(* IEC 61131-3 sources: ATCMcontrol_Engineering/src/COM/softing/fc/CL/Libs/ATCM_IEC1131_3, 277 files *)

(* ---- abs.st ---- *)
(*[[
    UserURL= "ATCMfile:ABS.htm"
]]*)

FUNCTION ABS : ANY_NUM
VAR_INPUT
    IN : ANY_NUM;
END_VAR

overload () inline{java.lang.Math.abs(%1)}

END_FUNCTION

(* ---- acos.st ---- *)
(*[[
    UserURL= "ATCMfile:ACOS.htm"
]]*)

FUNCTION ACOS : ANY_REAL
VAR_INPUT
    IN : ANY_REAL;
END_VAR

overload () inline{java.lang.Math.acos(%1)}

END_FUNCTION

(* ---- add.st ---- *)
(*[[
    UserURL= "ATCMFile:ADD.htm"
]]*)

FUNCTION ADD : ANY_MAGNITUDE
VAR_INPUT
    IN1 : ANY_MAGNITUDE;
END_VAR
VAR_IN_EXT
    IN2 : ANY_MAGNITUDE;
END_VAR

inline +

END_FUNCTION

(* ---- add_dt_time.st ---- *)
(*[[
    UserURL= "ATCMFile:ADD_DT_TIME.htm"
]]*)

FUNCTION ADD_DT_TIME : DT
VAR_INPUT
    IN1  : DT;
    IN2  : TIME;
END_VAR
inline +
END_FUNCTION

(* ---- add_time.st ---- *)
(*[[
    UserURL= "ATCMFile:ADD_TIME.htm"
]]*)

FUNCTION ADD_TIME : TIME
VAR_INPUT
    IN1 : TIME;
    IN2 : TIME;
END_VAR

inline +

END_FUNCTION

(* ---- add_tod_time.st ---- *)
(*[[
    UserURL= "ATCMFile:ADD_TOD_TIME.htm"
]]*)

FUNCTION ADD_TOD_TIME : TOD
VAR_INPUT
    IN1 : TOD;
    IN2 : TIME;
END_VAR
inline +
END_FUNCTION

(* ---- and.st ---- *)
(*[[
    UserURL= "ATCMFile:AND.htm"
]]*)

FUNCTION AND : ANY_BIT
VAR_INPUT
    IN1 : ANY_BIT;
END_VAR
VAR_IN_EXT
    IN2 : ANY_BIT;
END_VAR

inline AND

END_FUNCTION

(* ---- asin.st ---- *)
(*[[
    UserURL= "ATCMFile:ASIN.htm"
]]*)

FUNCTION ASIN : ANY_REAL
VAR_INPUT
    IN : ANY_REAL;
END_VAR

overload () inline{java.lang.Math.asin(%1)}

END_FUNCTION

(* ---- atan.st ---- *)
(*[[
    UserURL= "ATCMFile:ATAN.htm"
]]*)

FUNCTION ATAN : ANY_REAL
VAR_INPUT
    IN : ANY_REAL;
END_VAR

overload () inline{java.lang.Math.atan(%1)}

END_FUNCTION

(* ---- bool_to_byte.st ---- *)
(*[[
    UserURL= "ATCMFile:BOOL_TO_BYTE.htm"
]]*)

FUNCTION BOOL_TO_BYTE : BYTE
VAR_INPUT
    IN : BOOL;
END_VAR

inline{%1?1:0}

END_FUNCTION

(* ---- bool_to_dint.st ---- *)
(*[[
    UserURL= "ATCMFile:BOOL_TO_DINT.htm"
]]*)

FUNCTION BOOL_TO_DINT : DINT
VAR_INPUT
    IN : BOOL;
END_VAR

inline{%1?1:0}

END_FUNCTION

(* ---- bool_to_dword.st ---- *)
(*[[
    UserURL= "ATCMFile:BOOL_TO_DWORD.htm"
]]*)

FUNCTION BOOL_TO_DWORD : DWORD
VAR_INPUT
    IN : BOOL;
END_VAR

inline{%1?1:0}

END_FUNCTION

(* ---- bool_to_int.st ---- *)
(*[[
    UserURL= "ATCMFile:BOOL_TO_INT.htm"
]]*)

FUNCTION BOOL_TO_INT : INT
VAR_INPUT
    IN : BOOL;
END_VAR

inline{ VMOP(bool_to_int) }

END_FUNCTION

(* ---- bool_to_lint.st ---- *)
(*[[
    UserURL= "ATCMFile:BOOL_TO_LINT.htm"
]]*)

FUNCTION BOOL_TO_LINT : LINT
VAR_INPUT
    IN : BOOL;
END_VAR

inline{%1?1l:0l}

END_FUNCTION

(* ---- bool_to_lreal.st ---- *)
(*[[
    UserURL= "ATCMFile:BOOL_TO_LREAL.htm"
]]*)

FUNCTION BOOL_TO_LREAL : LREAL
VAR_INPUT
    IN : BOOL;
END_VAR

inline{%1?1.0:0.0}

END_FUNCTION

(* ---- bool_to_lword.st ---- *)
(*[[
    UserURL= "ATCMFile:BOOL_TO_LWORD.htm"
]]*)

FUNCTION BOOL_TO_LWORD : LWORD
VAR_INPUT
    IN : BOOL;
END_VAR

inline{%1?1l:0l}

END_FUNCTION

(* ---- bool_to_real.st ---- *)
(*[[
    UserURL= "ATCMFile:BOOL_TO_REAL.htm"
]]*)

FUNCTION BOOL_TO_REAL : REAL
VAR_INPUT
    IN : BOOL;
END_VAR

inline{ VMOP }

END_FUNCTION

(* ---- bool_to_string.st ---- *)
(*[[
    UserURL= "ATCMFile:BOOL_TO_STRING.htm"
]]*)

FUNCTION BOOL_TO_STRING : STRING
VAR_INPUT
    IN : BOOL;
END_VAR

inline{ STDLIB(bool_to_string) }

END_FUNCTION

(* ---- bool_to_udint.st ---- *)
(*[[
    UserURL= "ATCMFile:BOOL_TO_UDINT.htm"
]]*)
FUNCTION BOOL_TO_UDINT : UDINT
VAR_INPUT
    IN : BOOL;
END_VAR

inline{ VMOP }

END_FUNCTION

(* ---- bool_to_uint.st ---- *)
(*[[
    UserURL= "ATCMFile:BOOL_TO_UINT.htm"
]]*)
FUNCTION BOOL_TO_UINT : UINT
VAR_INPUT
    IN : BOOL;
END_VAR

inline{ VMOP }

END_FUNCTION

(* ---- bool_to_word.st ---- *)
(*[[
    UserURL= "ATCMFile:BOOL_TO_WORD.htm"
]]*)

FUNCTION BOOL_TO_WORD : WORD
VAR_INPUT
    IN : BOOL;
END_VAR

inline{%1?1:0}

END_FUNCTION

(* ---- bool_to_wstring.st ---- *)
(*[[
    UserURL= "ATCMFile:BOOL_TO_WSTRING.htm"
]]*)

FUNCTION BOOL_TO_WSTRING : WSTRING
VAR_INPUT
    IN : BOOL;
END_VAR

inline{%1?"TRUE":"FALSE"}

END_FUNCTION

(* ---- byte_to_bool.st ---- *)
(*[[
    UserURL= "ATCMFile:BYTE_TO_BOOL.htm"
]]*)

FUNCTION BYTE_TO_BOOL : BOOL
VAR_INPUT
    IN : BYTE;
END_VAR

inline{%1==0?false:true}

END_FUNCTION

(* ---- byte_to_dint.st ---- *)
(*[[
    UserURL= "ATCMFile:BYTE_TO_DINT.htm"
]]*)

FUNCTION BYTE_TO_DINT : DINT
VAR_INPUT
    IN : BYTE;
END_VAR

inline{%1}

END_FUNCTION

(* ---- byte_to_dword.st ---- *)
(*[[
    UserURL= "ATCMFile:BYTE_TO_DWORD.htm"
]]*)

FUNCTION BYTE_TO_DWORD : DWORD
VAR_INPUT
    IN : BYTE;
END_VAR

inline{%1}

END_FUNCTION

(* ---- byte_to_int.st ---- *)
(*[[
    UserURL= "ATCMFile:BYTE_TO_INT.htm"
]]*)

FUNCTION BYTE_TO_INT : INT
VAR_INPUT
    IN : BYTE;
END_VAR

inline{ VMOP }

END_FUNCTION

(* ---- byte_to_lint.st ---- *)
(*[[
    UserURL= "ATCMFile:BYTE_TO_LINT.htm"
]]*)

FUNCTION BYTE_TO_LINT : LINT
VAR_INPUT
    IN : BYTE;
END_VAR

inline{(long)%1}

END_FUNCTION

(* ---- byte_to_lreal.st ---- *)
(*[[
    UserURL= "ATCMFile:BYTE_TO_LREAL.htm"
]]*)

FUNCTION BYTE_TO_LREAL : LREAL
VAR_INPUT
    IN : BYTE;
END_VAR

inline{(double)%1}

END_FUNCTION

(* ---- byte_to_lword.st ---- *)
(*[[
    UserURL= "ATCMFile:BYTE_TO_LWORD.htm"
]]*)

FUNCTION BYTE_TO_LWORD : LWORD
VAR_INPUT
    IN : BYTE;
END_VAR

inline{(long)%1}

END_FUNCTION

(* ---- byte_to_real.st ---- *)
(*[[
    UserURL= "ATCMFile:BYTE_TO_REAL.htm"
]]*)

FUNCTION BYTE_TO_REAL : REAL
VAR_INPUT
    IN : BYTE;
END_VAR

inline{VMOP}

END_FUNCTION

(* ---- byte_to_string.st ---- *)
(*[[
    UserURL= "ATCMFile:BYTE_TO_STRING.htm"
]]*)

FUNCTION BYTE_TO_STRING : STRING
VAR_INPUT
    IN : BYTE;
END_VAR

inline{ STDLIB(byte_to_string) }

END_FUNCTION

(* ---- byte_to_udint.st ---- *)
(*[[
    UserURL= "ATCMFile:BYTE_TO_UDINT.htm"
]]*)
FUNCTION BYTE_TO_UDINT : UDINT
VAR_INPUT
    IN : BYTE;
END_VAR

inline{ VMOP }

END_FUNCTION

(* ---- byte_to_uint.st ---- *)
(*[[
    UserURL= "ATCMFile:BYTE_TO_UINT.htm"
]]*)
FUNCTION BYTE_TO_UINT : UINT
VAR_INPUT
    IN : BYTE;
END_VAR

inline{ VMOP }

END_FUNCTION

(* ---- byte_to_word.st ---- *)
(*[[
    UserURL= "ATCMFile:BYTE_TO_WORD.htm"
]]*)

FUNCTION BYTE_TO_WORD : WORD
VAR_INPUT
    IN : BYTE;
END_VAR

inline{%1}

END_FUNCTION

(* ---- byte_to_wstring.st ---- *)
(*[[
    UserURL= "ATCMFile:BYTE_TO_WSTRING.htm"
]]*)

FUNCTION BYTE_TO_WSTRING : WSTRING
VAR_INPUT
    IN : BYTE;
END_VAR

inline{java.lang.Integer.toString(%1)}

END_FUNCTION

(* ---- concat.st ---- *)
(*[[
    UserURL= "ATCMFile:CONCAT.htm"
]]*)

FUNCTION CONCAT : ANY_STRING
VAR_INPUT
    IN1 : ANY_STRING;
END_VAR
VAR_IN_EXT
    IN2 : ANY_STRING;
END_VAR

overload() inline {@+}

END_FUNCTION

(* ---- concat_date_tod.st ---- *)
(*[[
    UserURL= "ATCMFile:CONCAT_DATE_TOD.htm"
]]*)

FUNCTION CONCAT_DATE_TOD : DT
VAR_INPUT
    IN1 : DATE;
    IN2 : TOD;
END_VAR

inline{Utils.concat_date_tod(%1,%2)}

END_FUNCTION

(* ---- cos.st ---- *)
(*[[
    UserURL= "ATCMFile:COS.htm"
]]*)

FUNCTION COS : ANY_REAL
VAR_INPUT
    IN : ANY_REAL;
END_VAR

overload () inline{java.lang.Math.cos(%1)}

END_FUNCTION

(* ---- date_to_wstring.st ---- *)
(*[[
    UserURL= "ATCMFile:DATE_TO_WSTRING.htm"
]]*)

FUNCTION DATE_TO_WSTRING : WSTRING
VAR_INPUT
    IN : DATE;
END_VAR

inline{Utils.date_to_wstring(%1)}

END_FUNCTION

(* ---- delete.st ---- *)
(*[[
    UserURL= "ATCMFile:DELETE.htm"
]]*)

FUNCTION DELETE : ANY_STRING
VAR_INPUT
    IN : ANY_STRING;
    L : ANY_INT;
    P : ANY_INT;
END_VAR

overload STRING(STRING,INT,INT)
    inline{ STDLIB(DeleteString_int)}

overload STRING(STRING,DINT,DINT)
    inline{
        %res
        %2
        dint_to_int
        %3
        dint_to_int
        %1
        calfsys #DeleteString_int
		leave 8
        }

(*
overload STRING(STRING,LINT,LINT)
    inline{
        %res
        %2
        lint_to_int
        %3
        lint_to_int
        %1
        calfsys #DeleteString_int
	leave 12
        }

overload STRING(STRING,SINT,SINT)
    inline{
        %res
        %2
        sint_to_int
        %3
        sint_to_int
        %1
        calfsys #DeleteString_int
	leave 12
        }
*)

END_FUNCTION

(* ---- delete_dint.st ---- *)
(*[[
    UserURL= "ATCMFile:DELETE_DINT.htm"
]]*)

FUNCTION DELETE_DINT : ANY_STRING
VAR_INPUT
    IN : ANY_STRING;
    L  : DINT;
    P  : DINT;
END_VAR

overload() inline{Utils.deleteString(%1,%2,%3)}

END_FUNCTION

(* ---- dint_to_bool.st ---- *)
(*[[
    UserURL= "ATCMFile:DINT_TO_BOOL.htm"
]]*)

FUNCTION DINT_TO_BOOL : BOOL
VAR_INPUT
    IN : DINT;
END_VAR

inline{%1==0?false:true}

END_FUNCTION

(* ---- dint_to_byte.st ---- *)
(*[[
    UserURL= "ATCMFile:DINT_TO_BYTE.htm"
]]*)

FUNCTION DINT_TO_BYTE : BYTE
VAR_INPUT
    IN : DINT;
END_VAR

inline{%1&0xff}

END_FUNCTION

(* ---- dint_to_dword.st ---- *)
(*[[
    UserURL= "ATCMFile:DINT_TO_DWORD.htm"
]]*)

FUNCTION DINT_TO_DWORD : DWORD
VAR_INPUT
    IN : DINT;
END_VAR

inline{%1}

END_FUNCTION

(* ---- dint_to_int.st ---- *)
(*[[
    UserURL= "ATCMFile:DINT_TO_INT.htm"
]]*)

FUNCTION DINT_TO_INT : INT
VAR_INPUT
    IN : DINT;
END_VAR

inline{VMOP}

END_FUNCTION

(* ---- dint_to_lint.st ---- *)
(*[[
    UserURL= "ATCMFile:DINT_TO_LINT.htm"
]]*)

FUNCTION DINT_TO_LINT : LINT
VAR_INPUT
    IN : DINT;
END_VAR

inline{(long)%1}

END_FUNCTION

(* ---- dint_to_lreal.st ---- *)
(*[[
    UserURL= "ATCMFile:DINT_TO_LREAL.htm"
]]*)

FUNCTION DINT_TO_LREAL : LREAL
VAR_INPUT
    IN : DINT;
END_VAR

inline{(double)%1}

END_FUNCTION

(* ---- dint_to_lword.st ---- *)
(*[[
    UserURL= "ATCMFile:DINT_TO_LWORD.htm"
]]*)

FUNCTION DINT_TO_LWORD : LWORD
VAR_INPUT
    IN : DINT;
END_VAR

inline{(long)%1}

END_FUNCTION

(* ---- dint_to_real.st ---- *)
(*[[
    UserURL= "ATCMFile:DINT_TO_REAL.htm"
]]*)

FUNCTION DINT_TO_REAL : REAL
VAR_INPUT
    IN : DINT;
END_VAR

inline{VMOP}

END_FUNCTION

(* ---- dint_to_string.st ---- *)
(*[[
    UserURL= "ATCMFile:DINT_TO_STRING.htm"
]]*)

FUNCTION DINT_TO_STRING : STRING
VAR_INPUT
    IN : DINT;
END_VAR

inline{ STDLIB(dint_to_string) }

END_FUNCTION

(* ---- dint_to_time.st ---- *)
(*[[
    UserURL= "ATCMFile:DINT_TO_TIME.htm"
]]*)

FUNCTION DINT_TO_TIME : TIME
VAR_INPUT
    IN : DINT;
END_VAR

inline{(long)%1}

END_FUNCTION

(* ---- dint_to_udint.st ---- *)
(*[[
    UserURL= "ATCMFile:DINT_TO_UDINT.htm"
]]*)
FUNCTION DINT_TO_UDINT : UDINT
VAR_INPUT
    IN : DINT;
END_VAR

inline{NOOP}

END_FUNCTION

(* ---- dint_to_uint.st ---- *)
(*[[
    UserURL= "ATCMFile:DINT_TO_UINT.htm"
]]*)
FUNCTION DINT_TO_UINT : UINT
VAR_INPUT
    IN : DINT;
END_VAR

inline{ VMOP }

END_FUNCTION

(* ---- dint_to_word.st ---- *)
(*[[
    UserURL= "ATCMFile:DINT_TO_WORD.htm"
]]*)

FUNCTION DINT_TO_WORD : WORD
VAR_INPUT
    IN : DINT;
END_VAR

inline{%1&0xffff}

END_FUNCTION

(* ---- dint_to_wstring.st ---- *)
(*[[
    UserURL= "ATCMFile:DINT_TO_WSTRING.htm"
]]*)

FUNCTION DINT_TO_WSTRING : WSTRING
VAR_INPUT
    IN : DINT;
END_VAR

inline{java.lang.Integer.toString(%1)}

END_FUNCTION

(* ---- div.st ---- *)
(*[[
    UserURL= "ATCMFile:DIV.htm"
]]*)

FUNCTION DIV : ANY_NUM
VAR_INPUT
    IN1: ANY_NUM;
    IN2: ANY_NUM;
END_VAR

inline /

END_FUNCTION

(* ---- divtime.st ---- *)
(*[[
    UserURL= "ATCMFile:DIVTIME.htm"
]]*)

FUNCTION DIVTIME : TIME
VAR_INPUT
    IN1 : TIME;
    IN2 : ANY_NUM;
END_VAR

inline /

END_FUNCTION

(* ---- dt_to_date.st ---- *)
(*[[
    UserURL= "ATCMFile:DT_TO_DATE.htm"
]]*)

FUNCTION DT_TO_DATE : DATE
VAR_INPUT
    IN : DT;
END_VAR

inline{Utils.dt_to_date(%1)}

END_FUNCTION

(* ---- dt_to_time.st ---- *)
(*[[
    UserURL= "ATCMFile:DT_TO_TIME.htm"
]]*)

FUNCTION DT_TO_TIME : TIME
VAR_INPUT
    IN : DT;
END_VAR

inline{%1}

END_FUNCTION

(* ---- dt_to_tod.st ---- *)
(*[[
    UserURL= "ATCMFile:DT_TO_TOD.htm"
]]*)

FUNCTION DT_TO_TOD : TOD
VAR_INPUT
    IN : DT;
END_VAR

inline{Utils.dt_to_tod(%1)}

END_FUNCTION

(* ---- dt_to_wstring.st ---- *)
(*[[
    UserURL= "ATCMFile:DT_TO_WSTRING.htm"
]]*)

FUNCTION DT_TO_WSTRING : WSTRING
VAR_INPUT
    IN : DT;
END_VAR

inline{Utils.dt_to_wstring(%1)}

END_FUNCTION

(* ---- dword_to_bool.st ---- *)
(*[[
    UserURL= "ATCMFile:DWORD_TO_BOOL.htm"
]]*)

FUNCTION DWORD_TO_BOOL : BOOL
VAR_INPUT
    IN : DWORD;
END_VAR

inline{%1==0?false:true}

END_FUNCTION

(* ---- dword_to_byte.st ---- *)
(*[[
    UserURL= "ATCMFile:DWORD_TO_BYTE.htm"
]]*)

FUNCTION DWORD_TO_BYTE : BYTE
VAR_INPUT
    IN : DWORD;
END_VAR

inline{%1&0xff}

END_FUNCTION

(* ---- dword_to_dint.st ---- *)
(*[[
    UserURL= "ATCMFile:DWORD_TO_DINT.htm"
]]*)

FUNCTION DWORD_TO_DINT : DINT
VAR_INPUT
    IN : DWORD;
END_VAR

inline{%1}

END_FUNCTION

(* ---- dword_to_int.st ---- *)
(*[[
    UserURL= "ATCMFile:DWORD_TO_INT.htm"
]]*)

FUNCTION DWORD_TO_INT : INT
VAR_INPUT
    IN : DWORD;
END_VAR

inline{VMOP}

END_FUNCTION

(* ---- dword_to_lint.st ---- *)
(*[[
    UserURL= "ATCMFile:DWORD_TO_LINT.htm"
]]*)

FUNCTION DWORD_TO_LINT : LINT
VAR_INPUT
    IN : DWORD;
END_VAR

inline{((long)%1)&0xffffffffl}

END_FUNCTION

(* ---- dword_to_lreal.st ---- *)
(*[[
    UserURL= "ATCMFile:DWORD_TO_LREAL.htm"
]]*)

FUNCTION DWORD_TO_LREAL : LREAL
VAR_INPUT
    IN : DWORD;
END_VAR

inline{(double)(0x00000000ffffffffL & %1)}

END_FUNCTION

(* ---- dword_to_lword.st ---- *)
(*[[
    UserURL= "ATCMFile:DWORD_TO_LWORD.htm"
]]*)

FUNCTION DWORD_TO_LWORD : LWORD
VAR_INPUT
    IN : DWORD;
END_VAR

inline{((long)%1)&0xffffffffl}

END_FUNCTION

(* ---- dword_to_real.st ---- *)
(*[[
    UserURL= "ATCMFile:DWORD_TO_REAL.htm"
]]*)

FUNCTION DWORD_TO_REAL : REAL
VAR_INPUT
    IN : DWORD;
END_VAR

inline{VMOP}

END_FUNCTION

(* ---- dword_to_string.st ---- *)
(*[[
    UserURL= "ATCMFile:DWORD_TO_STRING.htm"
]]*)

FUNCTION DWORD_TO_STRING : STRING
VAR_INPUT
    IN : DWORD;
END_VAR

inline{ STDLIB(dword_to_string) }

END_FUNCTION

(* ---- dword_to_udint.st ---- *)
(*[[
    UserURL= "ATCMFile:DWORD_TO_UDINT.htm"
]]*)
FUNCTION DWORD_TO_UDINT : UDINT
VAR_INPUT
    IN : DWORD;
END_VAR

inline{NOOP}

END_FUNCTION

(* ---- dword_to_uint.st ---- *)
(*[[
    UserURL= "ATCMFile:DWORD_TO_UINT.htm"
]]*)
FUNCTION DWORD_TO_UINT : UINT
VAR_INPUT
    IN : DWORD;
END_VAR

inline{ VMOP }

END_FUNCTION

(* ---- dword_to_word.st ---- *)
(*[[
    UserURL= "ATCMFile:DWORD_TO_WORD.htm"
]]*)

FUNCTION DWORD_TO_WORD : WORD
VAR_INPUT
    IN : DWORD;
END_VAR

inline{%1&0xffff}

END_FUNCTION

(* ---- dword_to_wstring.st ---- *)
(*[[
    UserURL= "ATCMFile:DWORD_TO_WSTRING.htm"
]]*)

FUNCTION DWORD_TO_WSTRING : WSTRING
VAR_INPUT
    IN : DWORD;
END_VAR

inline{java.lang.Long.toString(0x00000000ffffffffL & %1)}

END_FUNCTION

(* ---- eq.st ---- *)
(*[[
    UserURL= "ATCMFile:EQ.htm"
]]*)

FUNCTION EQ : BOOL
VAR_INPUT
    IN1 : ANY_ELEMENTARY;
END_VAR
VAR_IN_EXT
    IN2 : ANY_ELEMENTARY;
END_VAR

inline =

END_FUNCTION

(* ---- exp.st ---- *)
(*[[
    UserURL= "ATCMFile:EXP.htm"
]]*)

FUNCTION EXP : ANY_REAL
VAR_INPUT
    IN : ANY_REAL;
END_VAR

overload () inline{java.lang.Math.exp(%1)}

END_FUNCTION

(* ---- expt.st ---- *)
(*[[
    UserURL= "ATCMFile:EXPT.htm"
]]*)

FUNCTION EXPT : ANY_REAL
VAR_INPUT
    IN1: ANY_REAL;
    IN2: ANY_NUM;
END_VAR

inline **

END_FUNCTION

(* ---- find.st ---- *)
(*[[
    UserURL= "ATCMFile:FIND.htm"
]]*)

FUNCTION FIND : ANY_INT
VAR_INPUT
    IN1 : ANY_STRING;
    IN2 : ANY_STRING;
END_VAR

overload INT(STRING,STRING)
    inline{ STDLIB(FindString_int) }

overload DINT(STRING,STRING)
    inline{
        %res
        dint_to_int
        %2
        %1
        calfsys #FindString_int
		leave 8
		int_to_dint
        }

(*
overload LINT(STRING,STRING)
    inline{
        %res
        lint_to_int
        %2
        %1
        calfsys #FindString_int
	leave 10
        }

overload SINT(STRING,STRING)
    inline{
        %res
        sint_to_int
        %2
        %1
        calfsys #FindString_int
	leave 10
        }
*)

END_FUNCTION

(* ---- find_dint.st ---- *)
(*[[
    UserURL= "ATCMFile:FIND_DINT.htm"
]]*)
FUNCTION FIND_DINT : DINT
VAR_INPUT
    IN1 : ANY_STRING;
    IN2 : ANY_STRING;
END_VAR

overload() inline{%1.indexOf(%2)+1}

END_FUNCTION

(* ---- ge.st ---- *)
(*[[
    UserURL= "ATCMFile:GE.htm"
]]*)

FUNCTION GE : BOOL
VAR_INPUT
    IN1 : ANY_ELEMENTARY;
END_VAR
VAR_IN_EXT
    IN2 : ANY_ELEMENTARY;
END_VAR

inline >=

END_FUNCTION

(* ---- gt.st ---- *)
(*[[
    UserURL= "ATCMFile:GT.htm"
]]*)

FUNCTION GT : BOOL
VAR_INPUT
    IN1 : ANY_ELEMENTARY;
END_VAR
VAR_IN_EXT
    IN2 : ANY_ELEMENTARY;
END_VAR

inline >

END_FUNCTION

(* ---- insert.st ---- *)
(*[[
    UserURL= "ATCMFile:INSERT.htm"
]]*)

FUNCTION INSERT : ANY_STRING
VAR_INPUT
    IN1 : ANY_STRING;
    IN2 : ANY_STRING;
    P : ANY_INT;
END_VAR

overload STRING(STRING,STRING,INT)
    inline{ STDLIB(InsertString_int)}

overload STRING(STRING,STRING,DINT)
    inline{
        %res
        %3
        dint_to_int
        %2
        %1
        calfsys #InsertString_int
		leave 10
        }

(*
overload STRING(STRING,STRING,LINT)
    inline{
        %res
        %3
        lint_to_int
        %2
        %1
        calfsys #InsertString_int
	leave 14
        }

overload STRING(STRING,STRING,SINT)
    inline{
        %res
        %3
        sint_to_int
        %2
        %1
        calfsys #InsertString_int
	leave 14
        }
*)

END_FUNCTION

(* ---- insert_dint.st ---- *)
(*[[
    UserURL= "ATCMFile:INSERT_DINT.htm"
]]*)

FUNCTION INSERT_DINT : ANY_STRING
VAR_INPUT
    IN1 : ANY_STRING;
    IN2 : ANY_STRING;
    P   : DINT;
END_VAR

overload() inline{Utils.insertString(%1,%2,%3)}

END_FUNCTION

(* ---- int_to_bool.st ---- *)
(*[[
    UserURL= "ATCMFile:INT_TO_BOOL.htm"
]]*)

FUNCTION INT_TO_BOOL : BOOL
VAR_INPUT
    IN : INT;
END_VAR

inline{VMOP(WORD_TO_BOOL)}

END_FUNCTION

(* ---- int_to_byte.st ---- *)
(*[[
    UserURL= "ATCMFile:INT_TO_BYTE.htm"
]]*)

FUNCTION INT_TO_BYTE : BYTE
VAR_INPUT
    IN : INT;
END_VAR

inline{VMOP(word_to_byte
; int_to_byte
; push word#16#ff
; and_word
)
      }

END_FUNCTION

(* ---- int_to_dint.st ---- *)
(*[[
    UserURL= "ATCMFile:INT_TO_DINT.htm"
]]*)

FUNCTION INT_TO_DINT : DINT
VAR_INPUT
    IN : INT;
END_VAR

inline{VMOP}

END_FUNCTION

(* ---- int_to_dword.st ---- *)
(*[[
    UserURL= "ATCMFile:INT_TO_DWORD.htm"
]]*)

FUNCTION INT_TO_DWORD : DWORD
VAR_INPUT
    IN : INT;
END_VAR

inline{VMOP}

END_FUNCTION

(* ---- int_to_lint.st ---- *)
(*[[
    UserURL= "ATCMFile:INT_TO_LINT.htm"
]]*)

FUNCTION INT_TO_LINT : LINT
VAR_INPUT
    IN : INT;
END_VAR

inline{VMOP}

END_FUNCTION

(* ---- int_to_lreal.st ---- *)
(*[[
    UserURL= "ATCMFile:INT_TO_LREAL.htm"
]]*)

FUNCTION INT_TO_LREAL : LREAL
VAR_INPUT
    IN : INT;
END_VAR

inline{VMOP}

END_FUNCTION

(* ---- int_to_real.st ---- *)
(*[[
    UserURL= "ATCMFile:INT_TO_REAL.htm"
]]*)

FUNCTION INT_TO_REAL : REAL
VAR_INPUT
    IN : INT;
END_VAR

inline{VMOP}

END_FUNCTION

(* ---- int_to_string.st ---- *)
(*[[
    UserURL= "ATCMFile:INT_TO_STRING.htm"
]]*)

FUNCTION INT_TO_STRING : STRING
VAR_INPUT
    IN : INT;
END_VAR

inline{ STDLIB(int_to_string) }

END_FUNCTION

(* ---- int_to_time.st ---- *)
(*[[
    UserURL= "ATCMFile:INT_TO_TIME.htm"
]]*)

FUNCTION INT_TO_TIME : TIME
VAR_INPUT
    IN : INT;
END_VAR

inline
{
	%1
	int_to_dint
}

END_FUNCTION

(* ---- int_to_udint.st ---- *)
(*[[
    UserURL= "ATCMFile:INT_TO_UDINT.htm"
]]*)
FUNCTION INT_TO_UDINT : UDINT
VAR_INPUT
    IN : INT;
END_VAR

inline{ VMOP }

END_FUNCTION

(* ---- int_to_uint.st ---- *)
(*[[
    UserURL= "ATCMFile:INT_TO_UINT.htm"
]]*)
FUNCTION INT_TO_UINT : UINT
VAR_INPUT
    IN : INT;
END_VAR

inline{NOOP}

END_FUNCTION

(* ---- int_to_word.st ---- *)
(*[[
    UserURL= "ATCMFile:INT_TO_WORD.htm"
]]*)

FUNCTION INT_TO_WORD : WORD
VAR_INPUT
    IN : INT;
END_VAR

inline{NOOP}

END_FUNCTION

(* ---- le.st ---- *)
(*[[
    UserURL= "ATCMFile:LE.htm"
]]*)

FUNCTION LE : BOOL
VAR_INPUT
    IN1 : ANY_ELEMENTARY;
END_VAR
VAR_IN_EXT
    IN2 : ANY_ELEMENTARY;
END_VAR

inline <=

END_FUNCTION

(* ---- left.st ---- *)
(*[[
    UserURL= "ATCMFile:LEFT.htm"
]]*)
FUNCTION LEFT : ANY_STRING
VAR_INPUT
    IN : ANY_STRING;
    L : ANY_INT;
END_VAR

overload STRING(STRING,INT)
    inline{ STDLIB(LeftString_int) }

overload STRING(STRING,DINT)
    inline{
        %res
        %2
        dint_to_int
        %1
        calfsys #LeftString_int
		leave 6
        }

(*
overload STRING(STRING,LINT)
    inline{
        %res
        %2
        lint_to_int
        %1
        calfsys #LeftString_int
        leave 10
        }

overload STRING(STRING,SINT)
    inline{
        %res
        %2
        sint_to_int
        %1
        calfsys #LeftString_int
        leave 10
        }
*)

END_FUNCTION

(* ---- left_dint.st ---- *)
(*[[
    UserURL= "ATCMFile:LEFT_DINT.htm"
]]*)

FUNCTION LEFT_DINT : ANY_STRING
VAR_INPUT
    IN : ANY_STRING;
    L  : DINT;
END_VAR

overload() inline{%1.substring(0,%2)}

END_FUNCTION

(* ---- len.st ---- *)
(*[[
    UserURL= "ATCMFile:LEN.htm"
]]*)
FUNCTION LEN : ANY_INT
VAR_INPUT
    IN : STRING;
END_VAR

overload INT(STRING) inline { STDLIB(strlen_int) }
overload DINT(STRING) inline
{
	%res
	%1
    calfsys #strlen_int %leave
    int_to_dint
}

END_FUNCTION

(* ---- len_dint.st ---- *)
(*[[
    UserURL= "ATCMFile:LEN_DINT.htm"
]]*)

FUNCTION LEN_DINT : DINT
VAR_INPUT
    IN : ANY_STRING;
END_VAR

overload() inline{%1.length()}

END_FUNCTION

(* ---- limit.st ---- *)
(*[[
    UserURL= "ATCMFile:LIMIT.htm"
]]*)

FUNCTION LIMIT : ANY_ELEMENTARY
VAR_INPUT
    MN : ANY_ELEMENTARY;
    IN : ANY_ELEMENTARY;
    MX : ANY_ELEMENTARY;
END_VAR

overload DINT|LINT|LREAL|TIME|ANY_DATE|BYTE|WORD(
         DINT|LINT|LREAL|TIME|ANY_DATE|BYTE|WORD,
         DINT|LINT|LREAL|TIME|ANY_DATE|BYTE|WORD,
         DINT|LINT|LREAL|TIME|ANY_DATE|BYTE|WORD)       inline{Math.min(Math.max(%2,%1),%3)}

overload DWORD(DWORD, DWORD, DWORD)                     inline{Utils.minDword(Utils.maxDword(%2,%1),%3)}
overload LWORD(LWORD, LWORD, LWORD)                     inline{Utils.minLword(Utils.maxLword(%2,%1),%3)}
overload ANY_STRING(ANY_STRING, ANY_STRING, ANY_STRING) inline{Utils.minString(Utils.maxString(%2,%1),%3)}
overload BOOL(BOOL, BOOL, BOOL)                         inline{(%2||%1) && %3}

END_FUNCTION

(* ---- lint_to_bool.st ---- *)
(*[[
    UserURL= "ATCMFile:LINT_TO_BOOL.htm"
]]*)

FUNCTION LINT_TO_BOOL : BOOL
VAR_INPUT
    IN : LINT;
END_VAR

inline{%1==0l?false:true}

END_FUNCTION

(* ---- lint_to_byte.st ---- *)
(*[[
    UserURL= "ATCMFile:LINT_TO_BYTE.htm"
]]*)

FUNCTION LINT_TO_BYTE : BYTE
VAR_INPUT
    IN : LINT;
END_VAR

inline{(int)%1&0xff}

END_FUNCTION

(* ---- lint_to_dint.st ---- *)
(*[[
    UserURL= "ATCMFile:LINT_TO_DINT.htm"
]]*)

FUNCTION LINT_TO_DINT : DINT
VAR_INPUT
    IN : LINT;
END_VAR

inline{(int)%1}

END_FUNCTION

(* ---- lint_to_dword.st ---- *)
(*[[
    UserURL= "ATCMFile:LINT_TO_DWORD.htm"
]]*)

FUNCTION LINT_TO_DWORD : DWORD
VAR_INPUT
    IN : LINT;
END_VAR

inline{(int)%1}

END_FUNCTION

(* ---- lint_to_int.st ---- *)
(*[[
    UserURL= "ATCMFile:LINT_TO_INT.htm"
]]*)

FUNCTION LINT_TO_INT : INT
VAR_INPUT
    IN : LINT;
END_VAR

inline{(int)%1}

END_FUNCTION

(* ---- lint_to_lreal.st ---- *)
(*[[
    UserURL= "ATCMFile:LINT_TO_LREAL.htm"
]]*)

FUNCTION LINT_TO_LREAL : LREAL
VAR_INPUT
    IN : LINT;
END_VAR

inline{(double)%1}

END_FUNCTION

(* ---- lint_to_lword.st ---- *)
(*[[
    UserURL= "ATCMFile:LINT_TO_LWORD.htm"
]]*)

FUNCTION LINT_TO_LWORD : LWORD
VAR_INPUT
    IN : LINT;
END_VAR

inline{%1}

END_FUNCTION

(* ---- lint_to_real.st ---- *)
(*[[
    UserURL= "ATCMFile:LINT_TO_REAL.htm"
]]*)

FUNCTION LINT_TO_REAL : REAL
VAR_INPUT
    IN : LINT;
END_VAR

inline{(double)%1}

END_FUNCTION

(* ---- lint_to_string.st ---- *)
(*[[
    UserURL= "ATCMFile:LINT_TO_STRING.htm"
]]*)

FUNCTION LINT_TO_STRING : STRING
VAR_INPUT
    IN : LINT;
END_VAR

inline{java.lang.Long.toString(%1)}

END_FUNCTION

(* ---- lint_to_time.st ---- *)
(*[[
    UserURL= "ATCMFile:LINT_TO_TIME.htm"
]]*)

FUNCTION LINT_TO_TIME : TIME
VAR_INPUT
    IN : LINT;
END_VAR

inline{%1}

END_FUNCTION

(* ---- lint_to_word.st ---- *)
(*[[
    UserURL= "ATCMFile:LINT_TO_WORD.htm"
]]*)

FUNCTION LINT_TO_WORD : WORD
VAR_INPUT
    IN : LINT;
END_VAR

inline{(int)%1&0xffff}

END_FUNCTION

(* ---- lint_to_wstring.st ---- *)
(*[[
    UserURL= "ATCMFile:LINT_TO_WSTRING.htm"
]]*)

FUNCTION LINT_TO_WSTRING : WSTRING
VAR_INPUT
    IN : LINT;
END_VAR

inline{java.lang.Long.toString(%1)}

END_FUNCTION

(* ---- ln.st ---- *)
(*[[
    UserURL= "ATCMFile:LN.htm"
]]*)

FUNCTION LN : ANY_REAL
VAR_INPUT
    IN : ANY_REAL;
END_VAR

overload () inline{java.lang.Math.log(%1)}

END_FUNCTION

(* ---- log.st ---- *)
(*[[
    UserURL= "ATCMFile:LOG.htm"
]]*)

FUNCTION LOG : ANY_REAL
VAR_INPUT
    IN : ANY_REAL;
END_VAR

overload () inline{java.lang.Math.log(%1)/java.lang.Math.log(10)}

END_FUNCTION

(* ---- lreal_to_bool.st ---- *)
(*[[
    UserURL= "ATCMFile:LREAL_TO_BOOL.htm"
]]*)

FUNCTION LREAL_TO_BOOL : BOOL
VAR_INPUT
    IN : LREAL;
END_VAR

inline{%1==0.0?false:true}

END_FUNCTION

(* ---- lreal_to_byte.st ---- *)
(*[[
    UserURL= "ATCMFile:LREAL_TO_BYTE.htm"
]]*)

FUNCTION LREAL_TO_BYTE : BYTE
VAR_INPUT
    IN : LREAL;
END_VAR

inline{((int)Math.round(%1))&0xff}

END_FUNCTION

(* ---- lreal_to_dint.st ---- *)
(*[[
    UserURL= "ATCMFile:LREAL_TO_DINT.htm"
]]*)

FUNCTION LREAL_TO_DINT : DINT
VAR_INPUT
    IN : LREAL;
END_VAR

inline{Utils.doubleToIntIEC599(%1)}

END_FUNCTION

(* ---- lreal_to_dword.st ---- *)
(*[[
    UserURL= "ATCMFile:LREAL_TO_DWORD.htm"
]]*)

FUNCTION LREAL_TO_DWORD : DWORD
VAR_INPUT
    IN : LREAL;
END_VAR

inline{(int)Math.round(%1)}

END_FUNCTION

(* ---- lreal_to_int.st ---- *)
(*[[
    UserURL= "ATCMFile:LREAL_TO_INT.htm"
]]*)

FUNCTION LREAL_TO_INT : INT
VAR_INPUT
    IN : LREAL;
END_VAR

inline{VMOP}

END_FUNCTION

(* ---- lreal_to_lint.st ---- *)
(*[[
    UserURL= "ATCMFile:LREAL_TO_LINT.htm"
]]*)

FUNCTION LREAL_TO_LINT : LINT
VAR_INPUT
    IN : LREAL;
END_VAR

inline{Utils.doubleToLongIEC599(%1)}

END_FUNCTION

(* ---- lreal_to_lword.st ---- *)
(*
 * Note:
 *  LREAL_TO_LWORD(x) is the same as
 *  LINT_TO_LWORD(LREAL_TO_LINT(x))
 *
 *  e.g.  LREAL_TO_LWORD(-1.0E0) = 16#ffffffffffffffff;
 *)

FUNCTION LREAL_TO_LWORD : LWORD
VAR_INPUT
    IN : LREAL;
END_VAR

inline{Math.round(%1)}

END_FUNCTION

(* ---- lreal_to_real.st ---- *)
(*[[
    UserURL= "ATCMFile:LREAL_TO_REAL.htm"
]]*)

FUNCTION LREAL_TO_REAL : REAL
VAR_INPUT
    IN : LREAL;
END_VAR

inline{VMOP}

END_FUNCTION

(* ---- lreal_to_string.st ---- *)
(*[[
    UserURL= "ATCMFile:LREAL_TO_STRING.htm"
]]*)

FUNCTION LREAL_TO_STRING : STRING
VAR_INPUT
    IN : LREAL;
END_VAR

inline{ STDLIB(lreal_to_string)}

END_FUNCTION

(* ---- lreal_to_time.st ---- *)
(*[[
    UserURL= "ATCMFile:LREAL_TO_TIME.htm"
]]*)

FUNCTION LREAL_TO_TIME : TIME
VAR_INPUT
    IN : LREAL;
END_VAR

inline{(long)%1}

END_FUNCTION

(* ---- lreal_to_udint.st ---- *)
(*[[
    UserURL= "ATCMFile:LREAL_TO_UDINT.htm"
]]*)
FUNCTION LREAL_TO_UDINT : UDINT
VAR_INPUT
    IN : LREAL;
END_VAR

inline{ VMOP }

END_FUNCTION

(* ---- lreal_to_uint.st ---- *)
(*[[
    UserURL= "ATCMFile:LREAL_TO_UINT.htm"
]]*)
FUNCTION LREAL_TO_UINT : UINT
VAR_INPUT
    IN : LREAL;
END_VAR

inline{ VMOP }

END_FUNCTION

(* ---- lreal_to_word.st ---- *)
(*[[
    UserURL= "ATCMFile:LREAL_TO_WORD.htm"
]]*)

FUNCTION LREAL_TO_WORD : WORD
VAR_INPUT
    IN : LREAL;
END_VAR

inline{((int)Math.round(%1))&0xffff}

END_FUNCTION

(* ---- lreal_to_wstring.st ---- *)
(*[[
    UserURL= "ATCMFile:LREAL_TO_WSTRING.htm"
]]*)

FUNCTION LREAL_TO_WSTRING : WSTRING
VAR_INPUT
    IN : LREAL;
END_VAR

inline{java.lang.Double.toString(%1)}

END_FUNCTION

(* ---- lt.st ---- *)
(*[[
    UserURL= "ATCMFile:LT.htm"
]]*)

FUNCTION LT : BOOL
VAR_INPUT
    IN1 : ANY_ELEMENTARY;
END_VAR
VAR_IN_EXT
    IN2 : ANY_ELEMENTARY;
END_VAR

inline <

END_FUNCTION

(* ---- lword_to_bool.st ---- *)
(*[[
    UserURL= "ATCMFile:LWORD_TO_BOOL.htm"
]]*)

FUNCTION LWORD_TO_BOOL : BOOL
VAR_INPUT
    IN : LWORD;
END_VAR

inline{%1==0l?false:true}

END_FUNCTION

(* ---- lword_to_byte.st ---- *)
(*[[
    UserURL= "ATCMFile:LWORD_TO_BYTE.htm"
]]*)

FUNCTION LWORD_TO_BYTE : BYTE
VAR_INPUT
    IN : LWORD;
END_VAR

inline{(int)%1&0xff}

END_FUNCTION

(* ---- lword_to_dint.st ---- *)
(*[[
    UserURL= "ATCMFile:LWORD_TO_DINT.htm"
]]*)

FUNCTION LWORD_TO_DINT : DINT
VAR_INPUT
    IN : LWORD;
END_VAR

inline{(int)%1}

END_FUNCTION

(* ---- lword_to_dword.st ---- *)
(*[[
    UserURL= "ATCMFile:LWORD_TO_DWORD.htm"
]]*)

FUNCTION LWORD_TO_DWORD : DWORD
VAR_INPUT
    IN : LWORD;
END_VAR

inline{(int)%1}

END_FUNCTION

(* ---- lword_to_int.st ---- *)
(*[[
    UserURL= "ATCMFile:LWORD_TO_INT.htm"
]]*)

FUNCTION LWORD_TO_INT : INT
VAR_INPUT
    IN : LWORD;
END_VAR

inline{(int)%1}

END_FUNCTION

(* ---- lword_to_lint.st ---- *)
(*[[
    UserURL= "ATCMFile:LWORD_TO_LINT.htm"
]]*)

FUNCTION LWORD_TO_LINT : LINT
VAR_INPUT
    IN : LWORD;
END_VAR

inline{%1}

END_FUNCTION

(* ---- lword_to_lreal.st ---- *)
(*[[
    UserURL= "ATCMFile:LWORD_TO_LREAL.htm"
]]*)
(*
 * Note:
 *  LWORD_TO_LREAL(x) is the same as
 *  LINT_TO_LREAL(LWORD_TO_LINT(x))
 *
 *  e.g.  LWORD_TO_LREAL(16#ffffffffffffffff) = -1.0E0
 *)
FUNCTION LWORD_TO_LREAL : LREAL
VAR_INPUT
    IN : LWORD;
END_VAR

inline{(double)%1}

END_FUNCTION

(* ---- lword_to_real.st ---- *)
(*[[
    UserURL= "ATCMFile:LWORD_TO_REAL.htm"
]]*)

FUNCTION LWORD_TO_REAL : REAL
VAR_INPUT
    IN : LWORD;
END_VAR

inline{(double)%1}

END_FUNCTION

(* ---- lword_to_string.st ---- *)
(*[[
    UserURL= "ATCMFile:LWORD_TO_STRING.htm"
]]*)

FUNCTION LWORD_TO_STRING : STRING
VAR_INPUT
    IN : LWORD;
END_VAR

inline{ STDLIB(not yet implemented) }

END_FUNCTION

(* ---- lword_to_word.st ---- *)
(*[[
    UserURL= "ATCMFile:LWORD_TO_WORD.htm"
]]*)

FUNCTION LWORD_TO_WORD : WORD
VAR_INPUT
    IN : LWORD;
END_VAR

inline{(int)%1&0xffff}

END_FUNCTION

(* ---- lword_to_wstring.st ---- *)
(*[[
    UserURL= "ATCMFile:LWORD_TO_WSTRING.htm"
]]*)

FUNCTION LWORD_TO_WSTRING : WSTRING
VAR_INPUT
    IN : LWORD;
END_VAR

inline{Utils.lword_to_wstring(%1)}

END_FUNCTION

(* ---- max.st ---- *)
(*[[
    UserURL= "ATCMFile:MAX.htm"
]]*)

FUNCTION MAX : ANY_ELEMENTARY
VAR_INPUT
    IN1 : ANY_ELEMENTARY;
END_VAR
VAR_IN_EXT
    IN2 : ANY_ELEMENTARY;
END_VAR

overload DINT|LINT|LREAL|BYTE|WORD|TIME|ANY_DATE(
         DINT|LINT|LREAL|BYTE|WORD|TIME|ANY_DATE,
         DINT|LINT|LREAL|BYTE|WORD|TIME|ANY_DATE, ...) inline{@Math.max}
overload BOOL(BOOL, BOOL, ...)                         inline{@||}
overload DWORD(DWORD, DWORD, ...)                      inline{@Utils.maxDword}
overload LWORD(LWORD, LWORD, ...)                      inline{@Utils.maxLword}
overload ANY_STRING(ANY_STRING, ANY_STRING, ...)       inline{@Utils.maxString}

END_FUNCTION

(* ---- mid.st ---- *)
(*[[
    UserURL= "ATCMFile:MID.htm"
]]*)

FUNCTION MID : ANY_STRING
VAR_INPUT
    IN : ANY_STRING;
    L : ANY_INT;
    P : ANY_INT;
END_VAR

overload STRING(STRING,INT,INT)
    inline{ STDLIB(MidString_int) }

overload STRING(STRING,DINT,DINT)
    inline{
        %res
        %2
        dint_to_int
        %3
        dint_to_int
	    %1
        calfsys #MidString_int
		leave  8
        }

(*
overload STRING(STRING,LINT,LINT)
    inline{
        %res
        %2
        lint_to_int
        %3
        lint_to_int
	%1
        calfsys #MidString_int
        leave 12
        }

overload STRING(STRING,SINT,SINT)
    inline{
        %res
        %2
        sint_to_int
        %3
        sint_to_int
	%1
        calfsys #MidString_int
        leave 12
        }
*)

END_FUNCTION

(* ---- mid_dint.st ---- *)
(*[[
    UserURL= "ATCMFile:MID_DINT.htm"
]]*)

FUNCTION MID_DINT : ANY_STRING
VAR_INPUT
    IN : ANY_STRING;
    L  : DINT;
    P  : DINT;
END_VAR

overload() inline{Utils.midString(%1,%2,%3)}

END_FUNCTION

(* ---- min.st ---- *)
(*[[
    UserURL= "ATCMFile:MIN.htm"
]]*)

FUNCTION MIN : ANY_ELEMENTARY
VAR_INPUT
    IN1 : ANY_ELEMENTARY;
END_VAR
VAR_IN_EXT
    IN2 : ANY_ELEMENTARY;
END_VAR

overload DINT|LINT|LREAL|BYTE|WORD|TIME|ANY_DATE(
         DINT|LINT|LREAL|BYTE|WORD|TIME|ANY_DATE,
         DINT|LINT|LREAL|BYTE|WORD|TIME|ANY_DATE, ...) inline{@Math.min}
overload BOOL(BOOL,BOOL, ...)                          inline{@&&}
overload DWORD(DWORD, DWORD, ...)                      inline{@Utils.minDword}
overload LWORD(LWORD, LWORD, ...)                      inline{@Utils.minLword}
overload ANY_STRING(ANY_STRING, ANY_STRING, ...)       inline{@Utils.minString}

END_FUNCTION

(* ---- mod.st ---- *)
(*[[
    UserURL= "ATCMFile:MOD.htm"
]]*)

FUNCTION MOD : ANY_INT
VAR_INPUT
    IN1: ANY_INT;
    IN2: ANY_INT;
END_VAR

inline MOD

END_FUNCTION

(* ---- move.st ---- *)
(*[[
    UserURL= "ATCMFile:MOVE.htm"
]]*)

FUNCTION MOVE: ANY
VAR_INPUT
    In: ANY;
END_VAR

inline :=

END_FUNCTION

(* ---- mul.st ---- *)
(*[[
    UserURL= "ATCMFile:MUL.htm"
]]*)

FUNCTION MUL : ANY_NUM
VAR_INPUT
    IN1 : ANY_NUM;
END_VAR
VAR_IN_EXT
    IN2 : ANY_NUM;
END_VAR

inline *

END_FUNCTION

(* ---- multime.st ---- *)
(*[[
    UserURL= "ATCMFile:MULTIME.htm"
]]*)

FUNCTION MULTIME : TIME
VAR_INPUT
    IN1 : TIME;
    IN2 : ANY_NUM;
END_VAR

inline *

END_FUNCTION

(* ---- mux.st ---- *)
(*[[
    UserURL= "ATCMFile:MUX.htm"
]]*)

FUNCTION MUX : ANY
VAR_INPUT
   K : ANY_INT;
   IN0: ANY;
END_VAR
VAR_IN_EXT
   IN1: ANY;
END_VAR

(* optimized multiplexer for 2 values *)
overload BOOL(DINT, BOOL, BOOL)
inline{Utils.mux2_b(tc,%1,%2,%3)}

overload BYTE|WORD|DWORD|DINT|DATE|TOD(
                 DINT,
                 BYTE|WORD|DWORD|DINT|DATE|TOD,
                 BYTE|WORD|DWORD|DINT|DATE|TOD)
inline{Utils.mux2_i(tc,%1,%2,%3)}

overload LREAL(DINT, LREAL, LREAL)
inline{Utils.mux2_d(tc,%1,%2,%3)}

overload WSTRING(DINT, WSTRING, WSTRING)
inline{Utils.mux2_s(tc,%1,%2,%3)}

overload LINT|LWORD|TIME|DT(
                 DINT,
                 LINT|LWORD|TIME|DT,
                 LINT|LWORD|TIME|DT)
inline{Utils.mux2_l(tc,%1,%2,%3)}

overload QVT_BOOL(DINT, QVT_BOOL, QVT_BOOL)
inline{(QvtBoolValue)Utils.mux2_qvt(tc,%1,%2,%3)}

overload QVT_BYTE|QVT_WORD|QVT_DWORD|QVT_DINT(
                 DINT,
                 QVT_BYTE|QVT_WORD|QVT_DWORD|QVT_DINT,
                 QVT_BYTE|QVT_WORD|QVT_DWORD|QVT_DINT)
inline{(QvtIntValue)Utils.mux2_qvt(tc,%1,%2,%3)}

overload QVT_LREAL(DINT, QVT_LREAL, QVT_LREAL)
inline{(QvtDoubleValue)Utils.mux2_qvt(tc,%1,%2,%3)}

overload ANY_DERIVED(DINT, ANY_DERIVED, ANY_DERIVED)
inline{Utils.mux2_od(tc,%1,%2,%3)}

(* optimized multiplexer for 3 values *)
overload BOOL(DINT, BOOL, BOOL, BOOL)
inline{Utils.mux3_b(tc,%1,%2,%3,%4)}

overload BYTE|WORD|DWORD|DINT|DATE|TOD(
         DINT,
         BYTE|WORD|DWORD|DINT|DATE|TOD,
         BYTE|WORD|DWORD|DINT|DATE|TOD,
         BYTE|WORD|DWORD|DINT|DATE|TOD)
inline{Utils.mux3_i(tc,%1,%2,%3,%4)}

overload LREAL(DINT, LREAL, LREAL, LREAL)
inline{Utils.mux3_d(tc,%1,%2,%3,%4)}

overload WSTRING(DINT, WSTRING, WSTRING, WSTRING)
inline{Utils.mux3_s(tc,%1,%2,%3,%4)}

overload LINT|LWORD|TIME|DT(
         DINT,
         LINT|LWORD|TIME|DT,
         LINT|LWORD|TIME|DT,
         LINT|LWORD|TIME|DT)
inline{Utils.mux3_l(tc,%1,%2,%3,%4)}

overload QVT_BOOL(DINT, QVT_BOOL, QVT_BOOL, QVT_BOOL)
inline{(QvtBoolValue)Utils.mux3_qvt(tc,%1,%2,%3,%4)}

overload QVT_BYTE|QVT_WORD|QVT_DWORD|QVT_DINT(
         DINT,
         QVT_BYTE|QVT_WORD|QVT_DWORD|QVT_DINT,
         QVT_BYTE|QVT_WORD|QVT_DWORD|QVT_DINT,
         QVT_BYTE|QVT_WORD|QVT_DWORD|QVT_DINT)
inline{(QvtIntValue)Utils.mux3_qvt(tc,%1,%2,%3,%4)}

overload QVT_LREAL(DINT, QVT_LREAL, QVT_LREAL, QVT_LREAL)
inline{(QvtDoubleValue)Utils.mux3_qvt(tc,%1,%2,%3,%4)}

overload ANY_DERIVED(DINT, ANY_DERIVED, ANY_DERIVED, ANY_DERIVED)
inline{Utils.mux3_od(tc,%1,%2,%3,%4)}

(* non optimized multiplexer with up to 10 values *)
overload BOOL(DINT, BOOL, ...)
inline{Utils.mux_b(tc,%nargs-1,%1,%2,%3(false),%4(false),%5(false),%6(false),%7(false),%8(false),%9(false),%10(false),%11(false))}

overload BYTE|WORD|DWORD|DINT|DATE|TOD(DINT, BYTE|WORD|DWORD|DINT|DATE|TOD, ...)
inline{Utils.mux_i(tc,%nargs-1,%1,%2,%3(0),%4(0),%5(0),%6(0),%7(0),%8(0),%9(0),%10(0),%11(0))}

overload LREAL(DINT, LREAL, ...)
inline{Utils.mux_d(tc,%nargs-1,%1,%2,%3(0.0),%4(0.0),%5(0.0),%6(0.0),%7(0.0),%8(0.0),%9(0.0),%10(0.0),%11(0.0))}

overload WSTRING(DINT, WSTRING, ...)
inline{Utils.mux_s(tc,%nargs-1,%1,%2,%3(null),%4(null),%5(null),%6(null),%7(null),%8(null),%9(null),%10(null),%11(null))}

overload LINT|LWORD|TIME|DT(DINT, LINT|LWORD|TIME|DT, ...)
inline{Utils.mux_l(tc,%nargs-1,%1,%2,%3(0),%4(0),%5(0),%6(0),%7(0),%8(0),%9(0),%10(0),%11(0))}

overload QVT_BOOL(DINT, QVT_BOOL, ...)
inline{(QvtBoolValue)Utils.mux_qvt(tc,%nargs-1,%1,%2,%3(null),%4(null),%5(null),%6(null),%7(null),%8(null),%9(null),%10(null),%11(null))}

overload QVT_BYTE|QVT_WORD|QVT_DWORD|QVT_DINT(DINT, QVT_BYTE|QVT_WORD|QVT_DWORD|QVT_DINT, ...)
inline{(QvtIntValue)Utils.mux_qvt(tc,%nargs-1,%1,%2,%3(null),%4(null),%5(null),%6(null),%7(null),%8(null),%9(null),%10(null),%11(null))}

overload QVT_LREAL(DINT, QVT_LREAL, ...)
inline{(QvtDoubleValue)Utils.mux_qvt(tc,%nargs-1,%1,%2,%3(null),%4(null),%5(null),%6(null),%7(null),%8(null),%9(null),%10(null),%11(null))}

overload ANY_DERIVED(DINT, ANY_DERIVED, ...)
inline{Utils.mux_od(tc,%nargs-1,%1,%2,%3(null),%4(null),%5(null),%6(null),%7(null),%8(null),%9(null),%10(null),%11(null))}

END_FUNCTION

(* ---- ne.st ---- *)
(*[[
    UserURL= "ATCMFile:NE.htm"
]]*)

FUNCTION NE : BOOL
VAR_INPUT
    IN1 : ANY_ELEMENTARY;
    IN2 : ANY_ELEMENTARY;
END_VAR

inline <>

END_FUNCTION

(* ---- not.st ---- *)
(*[[
    UserURL= "ATCMFile:NOT.htm"
]]*)

FUNCTION NOT : ANY_BIT
VAR_INPUT
    IN : ANY_BIT;
END_VAR

inline NOT

END_FUNCTION

(* ---- or.st ---- *)
(*[[
    UserURL= "ATCMFile:OR.htm"
]]*)

FUNCTION OR : ANY_BIT
VAR_INPUT
    IN1 : ANY_BIT;
END_VAR
VAR_IN_EXT
    IN2 : ANY_BIT;
END_VAR

inline OR

END_FUNCTION

(* ---- real_to_bool.st ---- *)
(*[[
    UserURL= "ATCMFile:REAL_TO_BOOL.htm"
]]*)

FUNCTION REAL_TO_BOOL : BOOL
VAR_INPUT
    IN : REAL;
END_VAR

inline{VMOP}

END_FUNCTION

(* ---- real_to_byte.st ---- *)
(*[[
    UserURL= "ATCMFile:REAL_TO_BYTE.htm"
]]*)

FUNCTION REAL_TO_BYTE : BYTE
VAR_INPUT
    IN : REAL;
END_VAR

inline{VMOP}

END_FUNCTION

(* ---- real_to_dint.st ---- *)
(*[[
    UserURL= "ATCMFile:REAL_TO_DINT.htm"
]]*)

FUNCTION REAL_TO_DINT : DINT
VAR_INPUT
    IN : REAL;
END_VAR

inline{VMOP}

END_FUNCTION

(* ---- real_to_dword.st ---- *)
(*[[
    UserURL= "ATCMFile:REAL_TO_DWORD.htm"
]]*)

FUNCTION REAL_TO_DWORD : DWORD
VAR_INPUT
    IN : REAL;
END_VAR

inline{VMOP}

END_FUNCTION

(* ---- real_to_int.st ---- *)
(*[[
    UserURL= "ATCMFile:REAL_TO_INT.htm"
]]*)

FUNCTION REAL_TO_INT : INT
VAR_INPUT
    IN : REAL;
END_VAR

inline{VMOP}

END_FUNCTION

(* ---- real_to_lint.st ---- *)
(*[[
    UserURL= "ATCMFile:REAL_TO_LINT.htm"
]]*)

FUNCTION REAL_TO_LINT : LINT
VAR_INPUT
    IN : REAL;
END_VAR

inline{VMOP(not_yet_implem)}

END_FUNCTION

(* ---- real_to_lreal.st ---- *)
(*[[
    UserURL= "ATCMFile:REAL_TO_LREAL.htm"
]]*)

FUNCTION REAL_TO_LREAL : LREAL
VAR_INPUT
    IN : REAL;
END_VAR

inline{VMOP}

END_FUNCTION

(* ---- real_to_lword.st ---- *)
(*[[
    UserURL= "ATCMFile:REAL_TO_LWORD.htm"
]]*)

FUNCTION REAL_TO_LWORD : LWORD
VAR_INPUT
    IN : REAL;
END_VAR

inline{VMOP(not_yet_implem)}

END_FUNCTION

(* ---- real_to_string.st ---- *)
(*[[
    UserURL= "ATCMFile:REAL_TO_STRING.htm"
]]*)

FUNCTION REAL_TO_STRING : STRING
VAR_INPUT
    IN : REAL;
END_VAR

inline{ STDLIB(real_to_string) }

END_FUNCTION

(* ---- real_to_time.st ---- *)
(*[[
    UserURL= "ATCMFile:REAL_TO_TIME.htm"
]]*)

FUNCTION REAL_TO_TIME : TIME
VAR_INPUT
    IN : REAL;
END_VAR

inline
{
    %1
    real_to_dint
}

END_FUNCTION

(* ---- real_to_udint.st ---- *)
(*[[
    UserURL= "ATCMFile:REAL_TO_UDINT.htm"
]]*)
FUNCTION REAL_TO_UDINT : UDINT
VAR_INPUT
    IN : REAL;
END_VAR

inline{ VMOP }

END_FUNCTION

(* ---- real_to_uint.st ---- *)
(*[[
    UserURL= "ATCMFile:REAL_TO_UINT.htm"
]]*)
FUNCTION REAL_TO_UINT : UINT
VAR_INPUT
    IN : REAL;
END_VAR

inline{ VMOP }

END_FUNCTION

(* ---- real_to_word.st ---- *)
(*[[
    UserURL= "ATCMFile:REAL_TO_WORD.htm"
]]*)

FUNCTION REAL_TO_WORD : WORD
VAR_INPUT
    IN : REAL;
END_VAR

inline{VMOP}

END_FUNCTION

(* ---- replace.st ---- *)
(*[[
    UserURL= "ATCMFile:REPLACE.htm"
]]*)

FUNCTION REPLACE : ANY_STRING
VAR_INPUT
    IN1 : ANY_STRING;
    IN2 : ANY_STRING;
    L : ANY_INT;
    P : ANY_INT;
END_VAR

overload STRING(STRING,STRING,INT,INT)
    inline{ STDLIB(ReplaceString_int) }

overload STRING(STRING,STRING,DINT,DINT)
    inline{
        %res
        %3
        dint_to_int
        %4
        dint_to_int
        %2
        %1
        calfsys #ReplaceString_int
		leave  12
        }

(*
overload STRING(STRING,STRING,LINT,LINT)
    inline{
        %res
        %3
        lint_to_int
        %4
        lint_to_int
        %2
        %1
        calfsys #ReplaceString_int
	leave 16
        }

overload STRING(STRING,STRING,SINT,SINT)
    inline{
        %res
        %3
        sint_to_int
        %4
        sint_to_int
        %2
        %1
        calfsys #ReplaceString_int
	leave 16
        }
*)

END_FUNCTION

(* ---- replace_dint.st ---- *)
(*[[
    UserURL= "ATCMFile:REPLACE_DINT.htm"
]]*)

FUNCTION REPLACE_DINT : ANY_STRING
VAR_INPUT
    IN1 : ANY_STRING;
    IN2 : ANY_STRING;
    L   : DINT;
    P   : DINT;
END_VAR

overload() inline{Utils.replaceString(%1,%2,%3,%4)}

END_FUNCTION

(* ---- right.st ---- *)
(*[[
    UserURL= "ATCMFile:RIGHT.htm"
]]*)

FUNCTION RIGHT : ANY_STRING
VAR_INPUT
    IN : ANY_STRING;
    L : ANY_INT;
END_VAR

overload STRING(STRING,INT)
    inline{ STDLIB(RightString_int) }

overload STRING(STRING,DINT)
    inline{
        %res
        %2
        dint_to_int
        %1
        calfsys #RightString_int
		leave  6
        }

(*
overload STRING(STRING,LINT)
    inline{
        %res
        %2
        lint_to_int
        %1
        calfsys #RightString_int
	leave 10
        }

overload STRING(STRING,SINT)
    inline{
        %res
        %2
        sint_to_int
        %1
        calfsys #RightString_int
	leave 10
        }
*)

END_FUNCTION

(* ---- right_dint.st ---- *)
(*[[
    UserURL= "ATCMFile:RIGHT_DINT.htm"
]]*)

FUNCTION RIGHT_DINT : ANY_STRING
VAR_INPUT
    IN : ANY_STRING;
    L  : DINT;
END_VAR

overload() inline{Utils.rightString(%1,%2)}

END_FUNCTION

(* ---- rol.st ---- *)
(*[[
    UserURL= "ATCMFile:ROL.htm"
]]*)

FUNCTION ROL : ANY_BIT
VAR_INPUT
    IN : ANY_BIT;
    N  : ANY_INT;
END_VAR

overload BOOL(BOOL,DINT)   inline{%1}
overload BYTE(BYTE,DINT)   inline{Utils.rol(%1,%2,8)}
overload WORD(WORD,DINT)   inline{Utils.rol(%1,%2,16)}
overload DWORD(DWORD,DINT) inline{Utils.rol(%1,%2,32)}
overload LWORD(LWORD,DINT) inline{Utils.rol_l(%1,%2)}

END_FUNCTION

(* ---- ror.st ---- *)
(*[[
    UserURL= "ATCMFile:ROR.htm"
]]*)

FUNCTION ROR : ANY_BIT
VAR_INPUT
    IN : ANY_BIT;
    N  : ANY_INT;
END_VAR

overload BOOL(BOOL,DINT)   inline{%1}
overload BYTE(BYTE,DINT)   inline{Utils.ror(%1,%2,8)}
overload WORD(WORD,DINT)   inline{Utils.ror(%1,%2,16)}
overload DWORD(DWORD,DINT) inline{Utils.ror(%1,%2,32)}
overload LWORD(LWORD,DINT) inline{Utils.ror_l(%1,%2)}

END_FUNCTION

(* ---- sel.st ---- *)
(*[[
    UserURL= "ATCMFile:SEL.htm"
]]*)

FUNCTION SEL : ANY
VAR_INPUT
    G   : BOOL;
    IN0 : ANY;
    IN1 : ANY;
END_VAR

overload ANY(BOOL, ANY, ANY) inline{%1 ? %3 : %2}

END_FUNCTION

(* ---- shl.st ---- *)
(*[[
    UserURL= "ATCMFile:SHL.htm"
]]*)

FUNCTION SHL : ANY_BIT
VAR_INPUT
    IN : ANY_BIT;
    N  : ANY_INT;
END_VAR

overload BOOL(BOOL,DINT)   inline{Utils.shift_bool(%1,%2)}
overload BYTE(BYTE,DINT)   inline{Utils.shl(%1,%2,8)}
overload WORD(WORD,DINT)   inline{Utils.shl(%1,%2,16)}
overload DWORD(DWORD,DINT) inline{Utils.shl(%1,%2,32)}
overload LWORD(LWORD,DINT) inline{Utils.shl_l(%1,%2)}

END_FUNCTION

(* ---- shr.st ---- *)
(*[[
    UserURL= "ATCMFile:SHR.htm"
]]*)

FUNCTION SHR : ANY_BIT
VAR_INPUT
    IN : ANY_BIT;
    N  : ANY_INT;
END_VAR

overload BOOL (BOOL, DINT)   inline{Utils.shift_bool(%1,%2)}
overload BYTE (BYTE, DINT)   inline{Utils.shr(%1,%2,8)}
overload WORD (WORD, DINT)   inline{Utils.shr(%1,%2,16)}
overload DWORD(DWORD,DINT)   inline{Utils.shr(%1,%2,32)}
overload LWORD(LWORD,DINT)   inline{Utils.shr_l(%1,%2)}

END_FUNCTION

(* ---- sin.st ---- *)
(*[[
    UserURL= "ATCMFile:SIN.htm"
]]*)

FUNCTION SIN : ANY_REAL
VAR_INPUT
    IN : ANY_REAL;
END_VAR

overload () inline{java.lang.Math.sin(%1)}

END_FUNCTION

(* ---- sqrt.st ---- *)
(*[[
    UserURL= "ATCMFile:SQRT.htm"
]]*)

FUNCTION SQRT : ANY_REAL
VAR_INPUT
    IN : ANY_REAL;
END_VAR

overload () inline{java.lang.Math.sqrt(%1)}

END_FUNCTION

(* ---- string_to_bool.st ---- *)
(*[[
    UserURL= "ATCMFile:STRING_TO_BOOL.htm"
]]*)

FUNCTION STRING_TO_BOOL : BOOL
VAR_INPUT
    IN : STRING;
END_VAR

inline { STDLIB(string_to_bool) }

END_FUNCTION

(* ---- string_to_byte.st ---- *)
(*[[
    UserURL= "ATCMFile:STRING_TO_BYTE.htm"
]]*)

FUNCTION STRING_TO_BYTE : BYTE
VAR_INPUT
    IN : STRING;
END_VAR

inline{ STDLIB(string_to_byte) }

END_FUNCTION

(* ---- string_to_date.st ---- *)
(*[[
    UserURL= "ATCMFile:STRING_TO_DATE.htm"
]]*)

FUNCTION STRING_TO_DATE : DATE
VAR_INPUT
    IN : STRING;
END_VAR

inline{ STDLIB(string_to_date) }

END_FUNCTION

(* ---- string_to_dint.st ---- *)
(*[[
    UserURL= "ATCMFile:STRING_TO_DINT.htm"
]]*)

FUNCTION STRING_TO_DINT : DINT
VAR_INPUT
    IN : STRING;
END_VAR

inline{ STDLIB(string_to_dint) }

END_FUNCTION

(* ---- string_to_dt.st ---- *)
(*[[
    UserURL= "ATCMFile:STRING_TO_DT.htm"
]]*)

FUNCTION STRING_TO_DT : DT
VAR_INPUT
    IN : STRING;
END_VAR

inline{VMOP(not_yet_implem)}

END_FUNCTION

(* ---- string_to_dword.st ---- *)
(*[[
    UserURL= "ATCMFile:STRING_TO_DWORD.htm"
]]*)

FUNCTION STRING_TO_DWORD : DWORD
VAR_INPUT
    IN : STRING;
END_VAR

inline{ STDLIB(string_to_dword) }

END_FUNCTION

(* ---- string_to_int.st ---- *)
(*[[
    UserURL= "ATCMFile:STRING_TO_INT.htm"
]]*)

FUNCTION STRING_TO_INT : INT
VAR_INPUT
    IN : STRING;
END_VAR

inline{ STDLIB(string_to_int) }

END_FUNCTION

(* ---- string_to_lint.st ---- *)
(*[[
    UserURL= "ATCMFile:STRING_TO_LINT.htm"
]]*)

FUNCTION STRING_TO_LINT : LINT
VAR_INPUT
    IN : STRING;
END_VAR

inline{VMOP(not_yet_implem)}

END_FUNCTION

(* ---- string_to_lreal.st ---- *)
(*[[
    UserURL= "ATCMFile:STRING_TO_LREAL.htm"
]]*)

FUNCTION STRING_TO_LREAL : LREAL
VAR_INPUT
    IN : STRING;
END_VAR

inline{ STDLIB(string_to_lreal) }

END_FUNCTION

(* ---- string_to_lword.st ---- *)
(*[[
    UserURL= "ATCMFile:STRING_TO_LWORD.htm"
]]*)

FUNCTION STRING_TO_LWORD : LWORD
VAR_INPUT
    IN : STRING;
END_VAR

inline{VMOP(not_yet_implem)}

END_FUNCTION

(* ---- string_to_real.st ---- *)
(*[[
    UserURL= "ATCMFile:STRING_TO_REAL.htm"
]]*)

FUNCTION STRING_TO_REAL : REAL
VAR_INPUT
    IN : STRING;
END_VAR

inline{ STDLIB(string_to_real) }
END_FUNCTION

(* ---- string_to_time.st ---- *)
(*[[
    UserURL= "ATCMFile:STRING_TO_TIME.htm"
]]*)

FUNCTION STRING_TO_TIME : TIME
VAR_INPUT
    IN : STRING;
END_VAR

inline{VMOP(not_yet_implem)}

END_FUNCTION

(* ---- string_to_tod.st ---- *)
(*[[
    UserURL= "ATCMFile:STRING_TO_TOD.htm"
]]*)

FUNCTION STRING_TO_TOD : TOD
VAR_INPUT
    IN : STRING;
END_VAR

inline{VMOP(not_yet_implem)}

END_FUNCTION

(* ---- string_to_udint.st ---- *)
(*[[
    UserURL= "ATCMFile:STRING_TO_UDINT.htm"
]]*)
FUNCTION STRING_TO_UDINT : UDINT
VAR_INPUT
    IN : STRING;
END_VAR

inline{ STDLIB(string_to_dword) }

END_FUNCTION

(* ---- string_to_uint.st ---- *)
(*[[
    UserURL= "ATCMFile:STRING_TO_UINT.htm"
]]*)
FUNCTION STRING_TO_UINT : UINT
VAR_INPUT
    IN : STRING;
END_VAR

inline{ STDLIB(string_to_word) }

END_FUNCTION

(* ---- string_to_word.st ---- *)
(*[[
    UserURL= "ATCMFile:STRING_TO_WORD.htm"
]]*)

FUNCTION STRING_TO_WORD : WORD
VAR_INPUT
    IN : STRING;
END_VAR

inline{ STDLIB(string_to_word) }

END_FUNCTION

(* ---- sub.st ---- *)
(*[[
    UserURL= "ATCMFile:SUB.htm"
]]*)

FUNCTION SUB : ANY_MAGNITUDE
VAR_INPUT
    IN1: ANY_MAGNITUDE;
    IN2: ANY_MAGNITUDE;
END_VAR

inline -

END_FUNCTION

(* ---- sub_date_date.st ---- *)
(*[[
    UserURL= "ATCMFile:SUB_DATE_DATE.htm"
]]*)

FUNCTION SUB_DATE_DATE : TIME
VAR_INPUT
    IN1 : DATE;
    IN2 : DATE;
END_VAR

inline -

END_FUNCTION

(* ---- sub_dt_dt.st ---- *)
(*[[
    UserURL= "ATCMFile:SUB_DT_DT.htm"
]]*)

FUNCTION SUB_DT_DT : TIME
VAR_INPUT
    IN1 : DT;
    IN2 : DT;
END_VAR

inline -

END_FUNCTION

(* ---- sub_dt_time.st ---- *)
(*[[
    UserURL= "ATCMFile:SUB_DT_TIME.htm"
]]*)

FUNCTION SUB_DT_TIME : DT
VAR_INPUT
    IN1 : DT;
    IN2 : TIME;
END_VAR

inline -

END_FUNCTION

(* ---- sub_time.st ---- *)
(*[[
    UserURL= "ATCMFile:SUB_TIME.htm"
]]*)

FUNCTION SUB_TIME : TIME
VAR_INPUT
    IN1 : TIME;
    IN2 : TIME;
END_VAR

inline -

END_FUNCTION

(* ---- sub_tod_time.st ---- *)
(*[[
    UserURL= "ATCMFile:SUB_TOD_TIME.htm"
]]*)

FUNCTION SUB_TOD_TIME : TOD
VAR_INPUT
    IN1 : TOD;
    IN2 : TIME;
END_VAR

inline -

END_FUNCTION

(* ---- sub_tod_tod.st ---- *)
(*[[
    UserURL= "ATCMFile:SUB_TOD_TOD.htm"
]]*)

FUNCTION SUB_TOD_TOD : TIME
VAR_INPUT
    IN1 : TOD;
    IN2 : TOD;
END_VAR

inline -

END_FUNCTION

(* ---- tan.st ---- *)
(*[[
    UserURL= "ATCMFile:TAN.htm"
]]*)

FUNCTION TAN : ANY_REAL
VAR_INPUT
    IN : ANY_REAL;
END_VAR

overload () inline{java.lang.Math.tan(%1)}

END_FUNCTION

(* ---- time_to_dint.st ---- *)
(*[[
    UserURL= "ATCMFile:TIME_TO_DINT.htm"
]]*)

FUNCTION TIME_TO_DINT : DINT
VAR_INPUT
    IN : TIME;
END_VAR

inline{(int)%1}

END_FUNCTION

(* ---- time_to_dt.st ---- *)
(*[[
    UserURL= "ATCMFile:TIME_TO_DT.htm"
]]*)

FUNCTION TIME_TO_DT : DT
VAR_INPUT
    IN : TIME;
END_VAR

inline{%1}

END_FUNCTION

(* ---- time_to_int.st ---- *)
(*[[
    UserURL= "ATCMFile:TIME_TO_INT.htm"
]]*)

FUNCTION TIME_TO_INT : INT
VAR_INPUT
    IN : TIME;
END_VAR

inline
{
    %1
    dint_to_int
}

END_FUNCTION

(* ---- time_to_lint.st ---- *)
(*[[
    UserURL= "ATCMFile:TIME_TO_LINT.htm"
]]*)

FUNCTION TIME_TO_LINT : LINT
VAR_INPUT
    IN : TIME;
END_VAR

inline{%1}

END_FUNCTION

(* ---- time_to_lreal.st ---- *)
(*[[
    UserURL= "ATCMFile:TIME_TO_LREAL.htm"
]]*)

FUNCTION TIME_TO_LREAL : LREAL
VAR_INPUT
    IN : TIME;
END_VAR

inline{(double)%1}

END_FUNCTION

(* ---- time_to_real.st ---- *)
(*[[
    UserURL= "ATCMFile:TIME_TO_REAL.htm"
]]*)

FUNCTION TIME_TO_REAL : REAL
VAR_INPUT
    IN : TIME;
END_VAR

inline
{
    %1
    dint_to_real
}

END_FUNCTION

(* ---- time_to_string.st ---- *)
(*[[
    UserURL= "ATCMFile:TIME_TO_STRING.htm"
]]*)

FUNCTION TIME_TO_STRING : STRING
VAR_INPUT
   IN : TIME;
END_VAR

inline{ STDLIB(time32_to_string) }

END_FUNCTION

(* ---- time_to_wstring.st ---- *)
(*[[
    UserURL= "ATCMFile:TIME_TO_WSTRING.htm"
]]*)

FUNCTION TIME_TO_WSTRING : WSTRING
VAR_INPUT
   IN : TIME;
END_VAR

inline{"t#"+java.lang.Long.toString(%1)+"ms"}

END_FUNCTION

(* ---- tod_to_string.st ---- *)
(*[[
    UserURL= "ATCMFile:TOD_TO_STRING.htm"
]]*)

FUNCTION TOD_TO_STRING : STRING
VAR_INPUT
    IN : TOD;
END_VAR

inline{ STDLIB(not yet implented) }

END_FUNCTION

(* ---- tod_to_time.st ---- *)
(*[[
    UserURL= "ATCMFile:TOD_TO_TIME.htm"
]]*)

FUNCTION TOD_TO_TIME : TIME
VAR_INPUT
    IN : TOD;
END_VAR

inline{(long)%1}

END_FUNCTION

(* ---- tod_to_wstring.st ---- *)
(*[[
    UserURL= "ATCMFile:TOD_TO_WSTRING.htm"
]]*)

FUNCTION TOD_TO_WSTRING : WSTRING
VAR_INPUT
    IN : TOD;
END_VAR

inline{Utils.tod_to_wstring(%1)}

END_FUNCTION

(* ---- trunc.st ---- *)
(*[[
    UserURL= "ATCMFile:TRUNC.htm"
]]*)

FUNCTION TRUNC : ANY_INT
VAR_INPUT
    IN : ANY_REAL;
END_VAR

overload DINT(ANY_REAL) inline{(int)%1}
overload LINT(ANY_REAL) inline{(long)%1}

END_FUNCTION

(* ---- udint_to_bool.st ---- *)
(*[[
    UserURL= "ATCMFile:UDINT_TO_BOOL.htm"
]]*)
FUNCTION UDINT_TO_BOOL : BOOL
VAR_INPUT
    IN : UDINT;
END_VAR

inline{ VMOP }

END_FUNCTION

(* ---- udint_to_byte.st ---- *)
(*[[
    UserURL= "ATCMFile:UDINT_TO_BYTE.htm"
]]*)
FUNCTION UDINT_TO_BYTE : BYTE
VAR_INPUT
    IN : UDINT;
END_VAR

inline{ VMOP }

END_FUNCTION

(* ---- udint_to_dint.st ---- *)
(*[[
    UserURL= "ATCMFile:UDINT_TO_DINT.htm"
]]*)
FUNCTION UDINT_TO_DINT : DINT
VAR_INPUT
    IN : UDINT;
END_VAR

inline{NOOP}

END_FUNCTION

(* ---- udint_to_dword.st ---- *)
(*[[
    UserURL= "ATCMFile:UDINT_TO_DWORD.htm"
]]*)
FUNCTION UDINT_TO_DWORD : DWORD
VAR_INPUT
    IN : UDINT;
END_VAR

inline{NOOP}

END_FUNCTION

(* ---- udint_to_int.st ---- *)
(*[[
    UserURL= "ATCMFile:UDINT_TO_INT.htm"
]]*)
FUNCTION UDINT_TO_INT : INT
VAR_INPUT
    IN : UDINT;
END_VAR

inline{ VMOP }

END_FUNCTION

(* ---- udint_to_lreal.st ---- *)
(*[[
    UserURL= "ATCMFile:UDINT_TO_LREAL.htm"
]]*)
FUNCTION UDINT_TO_LREAL : LREAL
VAR_INPUT
    IN : UDINT;
END_VAR

inline{ VMOP }

END_FUNCTION

(* ---- udint_to_real.st ---- *)
(*[[
    UserURL= "ATCMFile:UDINT_TO_REAL.htm"
]]*)
FUNCTION UDINT_TO_REAL : REAL
VAR_INPUT
    IN : UDINT;
END_VAR

inline{ VMOP }

END_FUNCTION

(* ---- udint_to_string.st ---- *)
(*[[
    UserURL= "ATCMFile:UDINT_TO_STRING.htm"
]]*)
FUNCTION UDINT_TO_STRING : STRING
VAR_INPUT
    IN : UDINT;
END_VAR

inline{ STDLIB(dword_to_string) }

END_FUNCTION

(* ---- udint_to_word.st ---- *)
(*[[
    UserURL= "ATCMFile:UDINT_TO_WORD.htm"
]]*)
FUNCTION UDINT_TO_WORD : WORD
VAR_INPUT
    IN : UDINT;
END_VAR

inline{ VMOP }

END_FUNCTION

(* ---- uint_to_bool.st ---- *)
(*[[
    UserURL= "ATCMFile:UINT_TO_BOOL.htm"
]]*)
FUNCTION UINT_TO_BOOL : BOOL
VAR_INPUT
    IN : UINT;
END_VAR

inline{ VMOP }

END_FUNCTION

(* ---- uint_to_byte.st ---- *)
(*[[
    UserURL= "ATCMFile:UINT_TO_BYTE.htm"
]]*)
FUNCTION UINT_TO_BYTE : BYTE
VAR_INPUT
    IN : UINT;
END_VAR

inline{ VMOP }

END_FUNCTION

(* ---- uint_to_dint.st ---- *)
(*[[
    UserURL= "ATCMFile:UINT_TO_DINT.htm"
]]*)
FUNCTION UINT_TO_DINT : DINT
VAR_INPUT
    IN : UINT;
END_VAR

inline{ VMOP }

END_FUNCTION

(* ---- uint_to_dword.st ---- *)
(*[[
    UserURL= "ATCMFile:UINT_TO_DWORD.htm"
]]*)
FUNCTION UINT_TO_DWORD : DWORD
VAR_INPUT
    IN : UINT;
END_VAR

inline{ VMOP }

END_FUNCTION

(* ---- uint_to_int.st ---- *)
(*[[
    UserURL= "ATCMFile:UINT_TO_INT.htm"
]]*)
FUNCTION UINT_TO_INT : INT
VAR_INPUT
    IN : UINT;
END_VAR

inline{NOOP}

END_FUNCTION

(* ---- uint_to_lreal.st ---- *)
(*[[
    UserURL= "ATCMFile:UINT_TO_LREAL.htm"
]]*)
FUNCTION UINT_TO_LREAL : LREAL
VAR_INPUT
    IN : UINT;
END_VAR

inline{ VMOP }

END_FUNCTION

(* ---- uint_to_real.st ---- *)
(*[[
    UserURL= "ATCMFile:UINT_TO_REAL.htm"
]]*)
FUNCTION UINT_TO_REAL : REAL
VAR_INPUT
    IN : UINT;
END_VAR

inline{ VMOP }

END_FUNCTION

(* ---- uint_to_string.st ---- *)
(*[[
    UserURL= "ATCMFile:UINT_TO_STRING.htm"
]]*)
FUNCTION UINT_TO_STRING : STRING
VAR_INPUT
    IN : UINT;
END_VAR

inline{ STDLIB(word_to_string) }

END_FUNCTION

(* ---- uint_to_word.st ---- *)
(*[[
    UserURL= "ATCMFile:UINT_TO_WORD.htm"
]]*)
FUNCTION UINT_TO_WORD : WORD
VAR_INPUT
    IN : UINT;
END_VAR

inline{NOOP}

END_FUNCTION

(* ---- word_string.st ---- *)
(*[[
    UserURL= "ATCMFile:WORD_TO_WSTRING.htm"
]]*)

FUNCTION WORD_TO_STRING : STRING
VAR_INPUT
    IN : WORD;
END_VAR

inline{VMOP}

END_FUNCTION

(* ---- word_to_bool.st ---- *)
(*[[
    UserURL= "ATCMFile:WORD_TO_BOOL.htm"
]]*)

FUNCTION WORD_TO_BOOL : BOOL
VAR_INPUT
    IN : WORD;
END_VAR

inline{%1==0?false:true}

END_FUNCTION

(* ---- word_to_byte.st ---- *)
(*[[
    UserURL= "ATCMFile:WORD_TO_BYTE.htm"
]]*)

FUNCTION WORD_TO_BYTE : BYTE
VAR_INPUT
    IN : WORD;
END_VAR

inline{%1&0xff}

END_FUNCTION

(* ---- word_to_dint.st ---- *)
(*[[
    UserURL= "ATCMFile:WORD_TO_DINT.htm"
]]*)

FUNCTION WORD_TO_DINT : DINT
VAR_INPUT
    IN : WORD;
END_VAR

inline{%1}

END_FUNCTION

(* ---- word_to_dword.st ---- *)
(*[[
    UserURL= "ATCMFile:WORD_TO_DWORD.htm"
]]*)

FUNCTION WORD_TO_DWORD : DWORD
VAR_INPUT
    IN : WORD;
END_VAR

inline{%1}

END_FUNCTION

(* ---- word_to_int.st ---- *)
(*[[
    UserURL= "ATCMFile:WORD_TO_INT.htm"
]]*)

FUNCTION WORD_TO_INT : INT
VAR_INPUT
    IN : WORD;
END_VAR

inline{NOOP}

END_FUNCTION

(* ---- word_to_lint.st ---- *)
(*[[
    UserURL= "ATCMFile:WORD_TO_LINT.htm"
]]*)

FUNCTION WORD_TO_LINT : LINT
VAR_INPUT
    IN : WORD;
END_VAR

inline{(long)%1}

END_FUNCTION

(* ---- word_to_lreal.st ---- *)
(*[[
    UserURL= "ATCMFile:WORD_TO_LREAL.htm"
]]*)

FUNCTION WORD_TO_LREAL : LREAL
VAR_INPUT
    IN : WORD;
END_VAR

inline{(double)%1}

END_FUNCTION

(* ---- word_to_lword.st ---- *)
(*[[
    UserURL= "ATCMFile:WORD_TO_LWORD.htm"
]]*)

FUNCTION WORD_TO_LWORD : LWORD
VAR_INPUT
    IN : WORD;
END_VAR

inline{(long)%1}

END_FUNCTION

(* ---- word_to_real.st ---- *)
(*[[
    UserURL= "ATCMFile:WORD_TO_REAL.htm"
]]*)

FUNCTION WORD_TO_REAL : REAL
VAR_INPUT
    IN : WORD;
END_VAR

inline{VMOP}

END_FUNCTION

(* ---- word_to_string.st ---- *)
(*[[
    UserURL= "ATCMFile:WORD_TO_STRING.htm"
]]*)

FUNCTION WORD_TO_STRING : STRING
VAR_INPUT
    IN : WORD;
END_VAR

inline{ STDLIB(word_to_string) }

END_FUNCTION

(* ---- word_to_udint.st ---- *)
(*[[
    UserURL= "ATCMFile:WORD_TO_UDINT.htm"
]]*)
FUNCTION WORD_TO_UDINT : UDINT
VAR_INPUT
    IN : WORD;
END_VAR

inline{ VMOP }

END_FUNCTION

(* ---- word_to_uint.st ---- *)
(*[[
    UserURL= "ATCMFile:WORD_TO_UINT.htm"
]]*)
FUNCTION WORD_TO_UINT : UINT
VAR_INPUT
    IN : WORD;
END_VAR

inline{NOOP}

END_FUNCTION

(* ---- word_to_wstring.st ---- *)
(*[[
    UserURL= "ATCMFile:WORD_TO_WSTRING.htm"
]]*)

FUNCTION WORD_TO_WSTRING : WSTRING
VAR_INPUT
    IN : WORD;
END_VAR

inline{java.lang.Integer.toString(%1)}

END_FUNCTION

(* ---- wstring_to_bool.st ---- *)
(*[[
    UserURL= "ATCMFile:WSTRING_TO_BOOL.htm"
]]*)

FUNCTION WSTRING_TO_BOOL : BOOL
VAR_INPUT
    IN : WSTRING;
END_VAR

inline{Utils.wstring_to_bool(tc,%1)}

END_FUNCTION

(* ---- wstring_to_byte.st ---- *)
(*[[
    UserURL= "ATCMFile:WSTRING_TO_BYTE.htm"
]]*)

FUNCTION WSTRING_TO_BYTE : BYTE
VAR_INPUT
    IN : WSTRING;
END_VAR

inline{Utils.wstring_to_byte(tc,%1)}

END_FUNCTION

(* ---- wstring_to_date.st ---- *)
(*[[
    UserURL= "ATCMFile:WSTRING_TO_DATE.htm"
]]*)

FUNCTION WSTRING_TO_DATE : DATE
VAR_INPUT
    IN : WSTRING;
END_VAR

inline{Utils.wstring_to_date(tc,%1)}

END_FUNCTION

(* ---- wstring_to_dint.st ---- *)
(*[[
    UserURL= "ATCMFile:WSTRING_TO_DINT.htm"
]]*)

FUNCTION WSTRING_TO_DINT : DINT
VAR_INPUT
    IN : WSTRING;
END_VAR

inline{Utils.wstring_to_dint(tc,%1)}

END_FUNCTION

(* ---- wstring_to_dt.st ---- *)
(*[[
    UserURL= "ATCMFile:WSTRING_TO_DT.htm"
]]*)

FUNCTION WSTRING_TO_DT : DT
VAR_INPUT
    IN : WSTRING;
END_VAR

inline{Utils.wstring_to_dt(tc,%1)}

END_FUNCTION

(* ---- wstring_to_dword.st ---- *)
(*[[
    UserURL= "ATCMFile:WSTRING_TO_DWORD.htm"
]]*)

FUNCTION WSTRING_TO_DWORD : DWORD
VAR_INPUT
    IN : WSTRING;
END_VAR

inline{Utils.wstring_to_dword(tc,%1)}

END_FUNCTION

(* ---- wstring_to_lint.st ---- *)
(*[[
    UserURL= "ATCMFile:WSTRING_TO_LINT.htm"
]]*)

FUNCTION WSTRING_TO_LINT : LINT
VAR_INPUT
    IN : WSTRING;
END_VAR

inline{Utils.wstring_to_lint(tc,%1)}

END_FUNCTION

(* ---- wstring_to_lreal.st ---- *)
(*[[
    UserURL= "ATCMFile:WSTRING_TO_LREAL.htm"
]]*)

FUNCTION WSTRING_TO_LREAL : LREAL
VAR_INPUT
    IN : WSTRING;
END_VAR

inline{Utils.wstring_to_lreal(tc,%1)}

END_FUNCTION

(* ---- wstring_to_lword.st ---- *)
(*[[
    UserURL= "ATCMFile:WSTRING_TO_LWORD.htm"
]]*)

FUNCTION WSTRING_TO_LWORD : LWORD
VAR_INPUT
    IN : WSTRING;
END_VAR

inline{Utils.wstring_to_lword(tc,%1)}

END_FUNCTION

(* ---- wstring_to_time.st ---- *)
(*[[
    UserURL= "ATCMFile:WSTRING_TO_TIME.htm"
]]*)

FUNCTION WSTRING_TO_TIME : TIME
VAR_INPUT
    IN : WSTRING;
END_VAR

inline{Utils.wstring_to_time(tc,%1)}

END_FUNCTION

(* ---- wstring_to_tod.st ---- *)
(*[[
    UserURL= "ATCMFile:WSTRING_TO_TOD.htm"
]]*)

FUNCTION WSTRING_TO_TOD : TOD
VAR_INPUT
    IN : WSTRING;
END_VAR

inline{Utils.wstring_to_tod(tc,%1)}

END_FUNCTION

(* ---- wstring_to_word.st ---- *)
(*[[
    UserURL= "ATCMFile:WSTRING_TO_WORD.htm"
]]*)

FUNCTION WSTRING_TO_WORD : WORD
VAR_INPUT
    IN : WSTRING;
END_VAR

inline{Utils.wstring_to_word(tc,%1)}

END_FUNCTION

(* ---- xor.st ---- *)
(*[[
    UserURL= "ATCMFile:XOR.htm"
]]*)

FUNCTION XOR : ANY_BIT
VAR_INPUT
    IN1 : ANY_BIT;
END_VAR
VAR_IN_EXT
    IN2 : ANY_BIT;
END_VAR

inline XOR

END_FUNCTION

(* ---- ctd.st ---- *)
(*[[
    UserURL= "ATCMFile:CTD_INT.htm"
]]*)
(*
 *  IEC-1131-3 Standard Functionblock CTD for data type INT
 *  Purpose: Down Counter
 *)
FUNCTION_BLOCK CTD
VAR_INPUT  (* Inputs *)
    CD         : BOOL R_EDGE; (* count down if rising edge     *)
    LD         : BOOL;        (* if true, copy PV to CV        *)
    PV         : INT;         (* start value                   *)
END_VAR
VAR_OUTPUT (* Outputs *)
    Q          : BOOL;        (* TRUE if CV <= 0               *)
    CV         : INT;         (* counter output                *)
END_VAR

;(* add target specific implementation here *)

END_FUNCTION_BLOCK

(* ---- ctd_dint.st ---- *)
(*[[
    UserURL= "ATCMFile:CTD_DINT.htm"
]]*)
(*
 *  IEC-1131-3 Standard Functionblock CTD for data type DINT
 *  Purpose: Down Counter
 *)
FUNCTION_BLOCK CTD_DINT
VAR_INPUT  (* Inputs *)
    CD         : BOOL R_EDGE; (* count down if rising edge     *)
    LD         : BOOL;        (* if true, copy PV to CV        *)
    PV         : DINT;        (* start value                   *)
END_VAR
VAR_OUTPUT (* Outputs *)
    Q          : BOOL;        (* TRUE if CV <= 0               *)
    CV         : DINT;        (* counter output                *)
END_VAR

  IF LD THEN
	CV := PV;
  ELSIF CD AND (CV > FC_MIN_DINT) THEN
	CV:=CV-1;
  END_IF;

  Q := (CV <= 0);

END_FUNCTION_BLOCK

(* ---- ctd_dint_ex.st ---- *)
(*[[
    UserURL= "ATCMFile:CTD_DINT_EX.htm"
]]*)
(*
 *  IEC-1131-3 Standard Functionblock CTD for data type DINT
 *  Purpose: Down Counter with visualisation scaling parameters
 *)
FUNCTION_BLOCK CTD_DINT_EX
VAR_INPUT  (* Inputs *)
    CD         : BOOL R_EDGE; (* count down if rising edge     *)
    LD         : BOOL;        (* if true, copy PV to CV        *)
    PV         : DINT;        (* start value                   *)
END_VAR
VAR_INPUT  (* Parameters *)
    SCALEMIN   : DINT:=0;     (* minimum of scaling            *)
    SCALEMAX   : DINT:=100;   (* maximum of scaling            *)
END_VAR
VAR_OUTPUT (* Outputs *)
    Q          : BOOL;        (* TRUE if CV <= 0               *)
    CV         : DINT;        (* counter output                *)
    ERROR      : DINT;        (* error                         *)
END_VAR

ERROR := 0;
IF (SCALEMIN >= SCALEMAX) THEN
   ERROR:=-1;
END_IF;

IF LD THEN
   CV := PV;
ELSIF CD AND (CV > FC_MIN_DINT) THEN
   CV:=CV-1;
END_IF;

Q := (CV <= 0);

END_FUNCTION_BLOCK

(* ---- ctu.st ---- *)
(*[[
    UserURL= "ATCMFile:CTU_INT.htm"
]]*)
(*
 *  IEC-1131-3 Standard Functionblock CTU for data type INT
 *  Purpose: Up Counter
 *)
FUNCTION_BLOCK CTU
VAR_INPUT (* Inputs *)
    CU         : BOOL R_EDGE; (* count up if rising edge *)
    R          : BOOL;        (* if true,  CV to zero    *)
    PV         : INT;         (* end value               *)
END_VAR
VAR_OUTPUT (* Outputs *)
    Q          : BOOL;        (* TRUE if CV >= PV        *)
    CV         : INT;         (* counter output          *)
END_VAR

;(* add target specific implementation here *)

END_FUNCTION_BLOCK

(* ---- ctu_dint.st ---- *)
(*[[
    UserURL= "ATCMFile:CTU_DINT.htm"
]]*)
(*
 *  IEC-1131-3 Standard Functionblock CTU for data type DINT
 *  Purpose: Up Counter
 *)
FUNCTION_BLOCK CTU_DINT
VAR_INPUT (* Inputs *)
    CU         : BOOL R_EDGE; (* count up if rising edge *)
    R          : BOOL;        (* if true,  CV to zero    *)
    PV         : DINT;        (* end value               *)
END_VAR
VAR_OUTPUT (* Outputs *)
    Q          : BOOL;        (* TRUE if CV >= PV        *)
    CV         : DINT;        (* counter output          *)
END_VAR

  IF R THEN
	CV := 0;
  ELSIF CU AND (CV < FC_MAX_DINT) THEN
	CV:=CV+1;
  END_IF;

  Q := (CV >= PV);

END_FUNCTION_BLOCK

(* ---- ctu_dint_ex.st ---- *)
(*[[
    UserURL= "ATCMFile:CTU_DINT_EX.htm"
]]*)
(*
 *  IEC-1131-3 Standard Functionblock CTU for data type DINT
 *  Purpose: Up Counter with visualisation scaling parameters
 *)
FUNCTION_BLOCK CTU_DINT_EX
VAR_INPUT  (* Inputs *)
    CU         : BOOL R_EDGE; (* count up if rising edge *)
    R          : BOOL;        (* if true,  CV to zero    *)
    PV         : DINT;        (* end value               *)
END_VAR
VAR_INPUT  (* Parameters *)
    SCALEMIN   : DINT:=0;     (* minimum of scaling      *)
    SCALEMAX   : DINT:=100;   (* maximum of scaling      *)
END_VAR
VAR_OUTPUT (* Outputs *)
    Q          : BOOL;        (* TRUE if CV >= PV        *)
    CV         : DINT;        (* counter output          *)
    ERROR      : DINT;        (* error                   *)
END_VAR

ERROR := 0;
IF (SCALEMIN >= SCALEMAX) THEN
    ERROR:=-1;
END_IF;

IF R THEN
    CV := 0;
ELSIF CU AND (CV < FC_MAX_DINT) THEN
    CV:=CV+1;
END_IF;

Q := (CV >= PV);

END_FUNCTION_BLOCK

(* ---- ctud.st ---- *)
(*[[
    UserURL= "ATCMFile:ctud_int.htm"
]]*)
(*
 *  IEC-1131-3 Standard Functionblock CTUD for data type INT
 *  Purpose: Up/Down Counter
 *)
FUNCTION_BLOCK CTUD
VAR_INPUT (* Inputs *)
    CU         : BOOL R_EDGE; (* count up if rising edge   *)
    CD         : BOOL R_EDGE; (* count down if rising edge *)
    R          : BOOL;        (* Reset, set CV to 0        *)
    LD         : BOOL;        (* if true, copy PV to CV    *)
    PV         : INT;         (* start value               *)
END_VAR
VAR_OUTPUT (* Outputs *)
    QU         : BOOL;        (* TRUE if CV >= PV          *)
    QD         : BOOL;        (* TRUE if CV <= 0           *)
    CV         : INT;         (* counter output            *)
END_VAR

;(* add target specific implementation here *)

END_FUNCTION_BLOCK

(* ---- ctud_dint.st ---- *)
(*[[
    UserURL= "ATCMFile:CTUD_DINT.htm"
]]*)
(*
 *  IEC-1131-3 Standard Functionblock CTUD for data type DINT
 *  Purpose: Up/Down Counter
 *)
FUNCTION_BLOCK CTUD_DINT
VAR_INPUT (* Inputs *)
    CU         : BOOL R_EDGE; (* count up if rising edge   *)
    CD         : BOOL R_EDGE; (* count down if rising edge *)
    R          : BOOL;        (* Reset, set CV to 0        *)
    LD         : BOOL;        (* if true, copy PV to CV    *)
    PV         : DINT;        (* start value               *)
END_VAR
VAR_OUTPUT (* Outputs *)
    QU         : BOOL;        (* TRUE if CV >= PV          *)
    QD         : BOOL;        (* TRUE if CV <= 0           *)
    CV         : DINT;        (* counter output            *)
END_VAR

  IF R THEN
	CV := 0;
  ELSIF LD THEN
	CV := PV;
  ELSE
	IF NOT (CU AND CD) THEN
		IF CU AND (CV < FC_MAX_DINT) THEN
			CV:=CV+1;
		ELSIF CD AND (CV > FC_MIN_DINT) THEN
			CV := CV-1;
		END_IF;
	END_IF;
  END_IF;

  QU := (CV >= PV);
  QD := (CV <= 0);

END_FUNCTION_BLOCK

(* ---- ctud_dint_ex.st ---- *)
(*[[
    UserURL= "ATCMFile:CTUD_DINT_EX.htm"
]]*)
(*
 *  IEC-1131-3 Standard Functionblock CTUD for data type DINT
 *  Purpose: Up/Down Counter with visualisation scaling parameters
 *)
FUNCTION_BLOCK CTUD_DINT_EX
VAR_INPUT (* Inputs *)
    CU         : BOOL R_EDGE; (* count up if rising edge   *)
    CD         : BOOL R_EDGE; (* count down if rising edge *)
    R          : BOOL;        (* Reset, set CV to 0        *)
    LD         : BOOL;        (* if true, copy PV to CV    *)
    PV         : DINT;        (* start value               *)
END_VAR
VAR_INPUT (* Parameters *)
    SCALEMIN   : DINT:=0;     (* minimum of scaling *)
    SCALEMAX   : DINT:=100;   (* maximum of scaling *)
END_VAR
VAR_OUTPUT (* Outputs *)
    QU         : BOOL;        (* TRUE if CV >= PV   *)
    QD         : BOOL;        (* TRUE if CV <= 0    *)
    CV         : DINT;        (* counter output     *)
    ERROR      : DINT;        (* error              *)
END_VAR

ERROR := 0;
IF (SCALEMIN >= SCALEMAX) THEN
    ERROR:=-1;
END_IF;

IF R THEN
   CV := 0;
ELSIF LD THEN
   CV := PV;
ELSE
   IF NOT (CU AND CD) THEN
      IF CU AND (CV < FC_MAX_DINT) THEN
         CV:=CV+1;
      ELSIF CD AND (CV > FC_MIN_DINT) THEN
         CV := CV-1;
      END_IF;
   END_IF;
END_IF;

QU := (CV >= PV);
QD := (CV <= 0);

END_FUNCTION_BLOCK

(* ---- f_trig.st ---- *)
(*[[
    UserURL= "ATCMFile:F_TRIG.htm"
]]*)
FUNCTION_BLOCK F_TRIG
VAR_INPUT
	CLK: BOOL;
END_VAR
VAR_OUTPUT
	Q: BOOL;
END_VAR
VAR
	M: BOOL := TRUE;
END_VAR

Q := NOT CLK AND NOT M;
M := NOT CLK;

END_FUNCTION_BLOCK

(* ---- r_trig.st ---- *)
(*[[
    UserURL= "ATCMFile:R_TRIG.htm"
]]*)
FUNCTION_BLOCK R_TRIG
VAR_INPUT
	CLK: BOOL;
END_VAR
VAR_OUTPUT
	Q: BOOL;
END_VAR
VAR
	M: BOOL := FALSE;
END_VAR

Q := CLK AND NOT M;
M := CLK;

END_FUNCTION_BLOCK

(* ---- rs.st ---- *)
(*[[
    UserURL= "ATCMFile:RS.htm"
]]*)
FUNCTION_BLOCK RS
VAR_INPUT
   S  : BOOL;
   R1 : BOOL;
END_VAR
VAR_OUTPUT
   Q1 : BOOL;
END_VAR

 Q1 := NOT R1 AND (S OR Q1);

END_FUNCTION_BLOCK

(* ---- sr.st ---- *)
(*[[
    UserURL= "ATCMFile:SR.htm"
]]*)
FUNCTION_BLOCK SR
VAR_INPUT
   S1 : BOOL;
   R  : BOOL;
END_VAR
VAR_OUTPUT
   Q1 : BOOL;
END_VAR

  Q1 := (NOT R AND Q1) OR S1;

END_FUNCTION_BLOCK

(* ---- tof.st ---- *)
(*[[
    UserURL= "ATCMFile:TOF.htm"
]]*)

FUNCTION_BLOCK TOF

VAR_INPUT   (* Inputs *)
    IN : BOOL := FALSE; (* Input        *)
    PT : TIME := T#0s;  (* Preset time  *)
END_VAR

VAR_OUTPUT  (* Outputs *)
    Q  : BOOL := FALSE; (* FALSE if ET >= PT *)
    ET : TIME := T#0s;  (* Elapsed time      *)
END_VAR

VAR NON_RETAIN
    StartTime : TIME;
    Trig : BOOL := FALSE;
END_VAR

IF PT > T#0s THEN
    IF IN THEN
        Q := TRUE;
        ET := T#0s;
        Trig := FALSE;
    ELSIF NOT Trig THEN
        Trig := TRUE;
        StartTime := getTimeSinceSystemBoot();
    ELSIF Q THEN
        ET := getTimeSinceSystemBoot() - StartTime;
        IF ET >= PT THEN
            Q := FALSE;
            ET := PT;
        END_IF;
    END_IF;
ELSE
	(* error handling *)
    Q := IN;
    ET := T#0s;
    Trig := FALSE;
END_IF;

END_FUNCTION_BLOCK

(* ---- tof_ex.st ---- *)
(*[[
    UserURL= "ATCMFile:TOF_EX.htm"
]]*)

FUNCTION_BLOCK TOF_EX

VAR_INPUT   (* Inputs *)
    IN : BOOL := FALSE; (* Input        *)
    PT : TIME := T#0s;  (* Preset time  *)
END_VAR

VAR_INPUT (* Parameters *)
    SCALEMIN : DINT := 0;   (* minimum of scaling *)
    SCALEMAX : DINT := 100; (* maximum of scaling *)
END_VAR

VAR_OUTPUT  (* Outputs *)
    Q  : BOOL := FALSE; (* FALSE if ET >= PT *)
    ET : TIME := T#0s;  (* Elapsed time      *)
    ERROR : DINT;       (* Error             *)
END_VAR

VAR NON_RETAIN
    StartTime : TIME;
    Trig : BOOL := FALSE;
END_VAR

  ERROR := 0;
  IF (SCALEMIN >= SCALEMAX) THEN
     ERROR := -1;
  END_IF;

  IF PT > T#0s THEN
    IF IN THEN
        Q := TRUE;
        ET := T#0s;
        Trig := FALSE;
    ELSIF NOT Trig THEN
        Trig := TRUE;
        StartTime := getTimeSinceSystemBoot();
    ELSIF Q THEN
        ET := getTimeSinceSystemBoot() - StartTime;
        IF ET >= PT THEN
            Q := FALSE;
            ET := PT;
        END_IF;
    END_IF;
  ELSE
    (* error handling *)
    Q := IN;
    ET := T#0s;
    Trig := FALSE;
    ERROR := -1;
  END_IF;

END_FUNCTION_BLOCK

(* ---- ton.st ---- *)
(*[[
    UserURL= "ATCMFile:TON.htm"
]]*)
FUNCTION_BLOCK TON

VAR_INPUT   (* Inputs *)
    IN : BOOL := FALSE; (* Input        *)
    PT : TIME := T#0s;  (* Preset time 	*)
END_VAR

VAR_OUTPUT  (* Outputs *)
    Q  : BOOL := FALSE; (* TRUE if ET >= PT *)
    ET : TIME := T#0s;  (* Elapsed time     *)
END_VAR

VAR NON_RETAIN
    StartTime : TIME;
    Trig : BOOL := FALSE;
END_VAR

IF PT > T#0s THEN
    IF NOT IN THEN
        Q := FALSE;
        ET := T#0s;
		Trig := FALSE;
    ELSIF NOT Trig THEN
        Trig := TRUE;
        StartTime := getTimeSinceSystemBoot();
    ELSIF NOT Q THEN
        ET := getTimeSinceSystemBoot() - StartTime;
        IF ET >= PT THEN
            Q := TRUE;
            ET := PT;
        END_IF;
    END_IF;
ELSE
	(* error handling *)
    Q := IN;
    ET := T#0s;
    Trig := FALSE;
END_IF;

END_FUNCTION_BLOCK

(* ---- ton_ex.st ---- *)
(*[[
    UserURL= "ATCMFile:TON_EX.htm"
]]*)

FUNCTION_BLOCK TON_EX

VAR_INPUT   (* Inputs *)
    IN : BOOL := FALSE; (* Input        *)
    PT : TIME := T#0s;  (* Preset time 	*)
END_VAR

VAR_INPUT   (* Parameters *)
    SCALEMIN : DINT := 0;   (* minimum of scaling *)
    SCALEMAX : DINT := 100; (* maximum of scaling *)
END_VAR

VAR_OUTPUT  (* Outputs *)
    Q  : BOOL := FALSE; (* TRUE if ET >= PT *)
    ET : TIME := T#0s;  (* Elapsed time     *)
    ERROR : DINT;       (* error            *)
END_VAR

VAR NON_RETAIN
    StartTime : TIME;
    Trig : BOOL := FALSE;
END_VAR

  ERROR := 0;
  IF (SCALEMIN >= SCALEMAX) THEN
     ERROR := -1;
  END_IF;

  IF PT > T#0s THEN
    IF NOT IN THEN
        Q := FALSE;
        ET := T#0s;
        Trig := FALSE;
    ELSIF NOT Trig THEN
        Trig := TRUE;
        StartTime := getTimeSinceSystemBoot();
    ELSIF NOT Q THEN
        ET := getTimeSinceSystemBoot() - StartTime;
        IF ET >= PT THEN
            Q := TRUE;
            ET := PT;
        END_IF;
    END_IF;
  ELSE
    (* error handling *)
    Q := IN;
    ET := T#0s;
    Trig := FALSE;
    ERROR := -1;
  END_IF;

END_FUNCTION_BLOCK

(* ---- tp.st ---- *)
(*[[
    UserURL= "ATCMFile:TP.htm"
]]*)

FUNCTION_BLOCK TP

VAR_INPUT   (* Inputs *)
    IN : BOOL := FALSE; (* Input       *)
    PT : TIME := T#0s;  (* Preset time *)
END_VAR

VAR_OUTPUT  (* Outputs *)
    Q  : BOOL := FALSE; (* FALSE if ET >= PT    *)
    ET : TIME := T#0s;  (* Elapsed time         *)
END_VAR

VAR
    M         : BOOL := FALSE;
END_VAR

VAR NON_RETAIN
    Trig      : BOOL := FALSE;
    StartTime : TIME;
END_VAR

IF PT > T#0s THEN
    IF NOT Trig THEN
        Q := FALSE;
        IF IN AND NOT M THEN
            (* initilize function block *)
            (* get start time *)
            Trig := TRUE;
            StartTime := getTimeSinceSystemBoot();
            ET := T#0s;
            Q := TRUE;
        ELSIF NOT IN THEN
            ET := T#0s;
        END_IF;
    ELSE (* IF Trig *)
        (* get elapsed time *)
        ET := getTimeSinceSystemBoot() - Starttime;

        IF ET >= PT THEN (* time reached *)
            Trig := FALSE;
            Q := FALSE;
            IF NOT IN THEN
              ET := T#0s;
            ELSE
              ET := PT;
            END_IF;
        END_IF;
	END_IF;

ELSE
    (* error handling *)
    Q := FALSE;
    ET := T#0s;
    Trig := FALSE;
END_IF;

M := IN;

END_FUNCTION_BLOCK

(* ---- tp_ex.st ---- *)
(*[[
    UserURL= "ATCMFile:TP_EX.htm"
]]*)

FUNCTION_BLOCK TP_EX

VAR_INPUT   (* Inputs *)
    IN : BOOL := FALSE; (* Input       *)
    PT : TIME := T#0s;  (* Preset time *)
END_VAR

VAR_INPUT (* Parameters *)
    SCALEMIN : DINT := 0;   (* minimum of scaling *)
    SCALEMAX : DINT := 100; (* maximum of scaling *)
END_VAR

VAR_OUTPUT  (* Outputs *)
    Q  : BOOL := FALSE; (* FALSE if ET >= PT    *)
    ET : TIME := T#0s;  (* Elapsed time         *)
    ERROR : DINT;       (* Error                *)
END_VAR

VAR
    M         : BOOL := FALSE;
END_VAR

VAR NON_RETAIN
    Trig      : BOOL := FALSE;
    StartTime : TIME;
END_VAR

  ERROR := 0;
  IF (SCALEMIN >= SCALEMAX) THEN
     ERROR := -1;
  END_IF;

  IF PT > T#0s THEN
    IF NOT Trig THEN
        Q := FALSE;
        IF IN AND NOT M THEN
            (* initilize function block *)
            (* get start time *)
            Trig := TRUE;
            StartTime := getTimeSinceSystemBoot();
            ET := T#0s;
            Q := TRUE;
        ELSIF NOT IN THEN
            ET := T#0s;
        END_IF;
    ELSE (* IF Trig *)
        (* get elapsed time *)
        ET := getTimeSinceSystemBoot() - Starttime;

        IF ET >= PT THEN (* time reached *)
            Trig := FALSE;
            Q := FALSE;
            IF NOT IN THEN
              ET := T#0s;
            ELSE
              ET := PT;
            END_IF;
        END_IF;
	END_IF;

  ELSE
    (* error handling *)
    Q := FALSE;
    ET := T#0s;
    Trig := FALSE;
    ERROR := -1;
  END_IF;

  M := IN;

END_FUNCTION_BLOCK
